        -0.63798948327222038,-0.021960985394712317,0.0,0.0,0.0,0.0,0.0,0.0,1.0,0.0,0.0,-0.0,-0.0,-0.0,-0.0,-0.0,
        -0.0,-1.0,-0.0,0.62490021645747618,0.58505858013174883,0.027072082181883242,0.027610578309122807,
        0.026708907388227909,-0.37854052611351124,-0.027072082181883242,-0.026708907388227909,0.0,0.0,0.0,0.0,0.0,
        0.0,0.0,0.0,-0.0,-0.0,-0.0,-0.0,-0.0,-0.0,-1.0,-0.0,0.027265477962947069,0.55566222109490582,
        0.63798667601923609,0.029437135799321879,0.62488169574462793,-0.55566181651356428,-0.023469887537635192,
        -0.62488169574462793,-0.63798609648432814,0.0,0.0,0.0,0.0,0.0,0.0,1.0,0.0,-0.0,-0.0,-0.0,-0.0,-0.0,-0.0,
        -1.0,-0.0,0.63800507768378822,0.027011667529779945,0.027541181508898387,0.026637267215644224,
        -0.45692709004827581,-0.027011667529779945,-0.58505858013174894,-0.027541181508898383,-0.026637267215644224,
        0.0,0.0,0.0,0.0,0.0,0.0,0.0,0.0,-0.0,-0.0,-0.0,-0.0,-0.0,-0.0,-1.0,-0.0,0.026352061912650541,
        0.55566389422834717,0.62488507878410182,0.637989575133729,-0.55566389422834717,-0.02598312883534095,
        -0.62488507878410182,-0.0294371357993219,-0.63798957513372911,0.0,0.0,0.0,0.0,0.0,0.0,1.0,0.0,-0.0,-0.0,
        -0.0,-0.0,-0.0,-0.0,-1.0,-0.0,-0.55566424910285672,-0.027034185307057621,0.70224208707170055,
        0.024752136540096732,0.70251617195999394,0.022319435462106595,0.0,0.0,0.0,0.0,0.0,0.0,0.0,0.0,-0.0,-0.0,
        -0.0,-0.0,-0.0,-0.0,-1.0,-0.0,-0.70226225634217332,-0.3785405261135113,-0.70163518723474272,
        0.027105602758215112,0.027648865450003536,0.026748274296612785,-0.027105602758215112,-0.027648865450003533,
        -0.026748274296612785,0.0,0.0,0.0,0.0,0.0,0.0,1.0,0.0,0.0,0.0,-0.0,-0.0,-0.0,-0.0,-0.0,-0.0,-0.0,
        -0.55566222109490582,0.023637206391576536,0.015100165961297108,-1.0,-0.378540460951947,-0.02764886545000354,
        0.015207454024849647,0.0,0.0,0.0,0.0,0.0,0.0,1.0,0.0,-0.0,-0.0,-0.0,-0.0,-0.0,-0.0,-0.45692709004827575,
        -0.702534060267215,0.027090859530371859,0.70163518723474272,-0.026730661933064313,0.0,0.0,0.0,0.0,0.0,0.0,
        0.0,0.0,-0.0,-0.0,-0.0,-0.0,-0.0,-0.0,-0.0,-0.55566389422834728,0.029709944333287521,-1.0,
        -0.37854017792555505,-0.026748274296612796,0.0,0.0,0.0,0.0,0.0,0.0,1.0,0.0,0.0,-0.0,-0.0,-0.0,-0.0,-0.0,
        -0.0,-0.55566424910285672,0.027034185307057621,-1.0,-0.37851997948504351,0.70317323754735273,
        -0.02240967789339866,0.0,0.0,0.0,0.0,0.0,0.0,0.0,0.0,-0.0,-0.0,-0.0,-0.0,-0.0,-0.0,-0.0,
        -0.55566222109490582,0.027566488177000255,0.70223873149897853,-0.023637206391576546,-0.015100165961297143,
        0.0,0.0,0.0,0.0,0.0,0.0,-0.0,-0.0,-0.0,-0.0,-0.0,-0.0,-1.0,-0.55566389422834728,0.026662833272981429,
        0.70224253943268344,0.70251656286365771,-0.026190122699982339,-0.029709944333287511,0.0,0.0,0.0,0.0,0.0,0.0,
        0.0,-0.0,-0.0,-0.0,-0.0,-0.0,-0.0,-1.0,-0.0,-0.02706527731251647,-0.6248806237808493,-0.023656120772106486,
        0.378519539943052,0.70317018870025627,0.0,0.0,0.0,0.0,0.0,0.0,0.0,0.0,-0.0,-0.0,-0.0,-0.0,-0.0,-0.0,
        -0.02346980199155271,-0.024399835479656976,0.55566129015943833,0.6248806237808493,0.63798497169620461,
        0.01473301981127613,-0.55566129015943833,-0.6248806237808493,-0.63798497169620461,0.0,0.0,0.0,0.0,0.0,0.0,
        1.0,0.0,-0.0,-0.0,-0.0,-0.0,-0.0,-0.0,-0.027011667529779945,-0.63798948327222027,0.456923837504278,
        0.58504518410006956,0.024723646828030479,0.0,0.0,0.0,0.0,0.0,0.0,1.0,0.0,-0.0,-0.0,-0.0,-0.0,-0.0,-0.0,-0.0,
        -0.02598312883534095,-0.021960985394712324,0.63798532239475636,-0.55566147407010114,-0.62488096344828059,
        -0.63798532239475636,0.0,0.0,0.0,0.0,0.0,0.0,1.0,0.0,0.0,0.0,-0.0,-0.0,-0.0,-0.0,-0.0,-0.0,-1.0,
        -0.027034185307057618,0.55566424910285683,0.024752136540096732,-0.70224208707170055,-0.70251617195999394,
        0.0,0.0,0.0,0.0,0.0,0.0,1.0,0.0,-0.0,-0.0,-0.0,-0.0,-0.0,-0.0,-0.0,-0.0,-0.02706527731251647,
        0.62488504774223075,0.024795740829694754,-0.37851997948504357,-0.7031738370963756,0.0,0.0,0.0,0.0,0.0,0.0,
        0.0,-0.0,-0.0,-0.0,-0.0,-0.0,-0.0,-0.0,-0.027011667529779945,0.63798948327222038,0.024723646828030479,
        0.02229166073122648,-0.456923837504278,-0.58504518410006945,0.0,0.0,0.0,0.0,0.0,0.0,0.0,-0.0,-0.0,-0.0,-0.0,
        -0.0,-0.0,-1.0,-0.0,-0.6248822663250807,-0.0276027315782233,-0.58504257002809312,-0.02974148887250478,
        0.37854036201549385,0.023660396850780661,0.0,0.0,0.0,0.0,0.0,0.0,1.0,0.0,-0.0,-0.0,-0.0,-0.0,-0.0,-0.0,
        -0.62488507878410182,-0.026700746627905073,-0.58504502721143925,0.37854017792555522,0.029748443430697026,
        0.0,0.0,0.0,0.0,0.0,0.0,1.0,0.0,-0.0,-0.0,-0.0,-0.0,-0.0,-0.0,-0.62488504774223086,-0.022364818883998015,
        -0.58504518410006956,0.027072082181883231,0.37854107343057747,-0.024805000972806229,0.0,0.0,0.0,0.0,0.0,0.0,
        1.0,0.0,-0.0,-0.0,-0.0,-0.0,-0.0,-0.0,-0.0,-0.58504257002809312,0.027610578309122814,0.37854046095194716,
        -0.023660296965944735,-0.015161281241640749,0.0,0.0,0.0,0.0,0.0,-0.0,-0.0,-0.0,-0.0,-0.0,
        -0.027541181508898383,-0.637986676019236,-0.029685529684818829,0.023621944154890266,0.58504204394174086,0.0,
        0.0,0.0,0.0,0.0,0.0,1.0,0.0,-0.0,-0.0,-0.0,-0.0,-0.0,-0.0,-0.027566488177000262,-0.70251319697861081,
        -0.029709944333287532,0.55566181651356417,0.023637304191565071,-0.70223802681964376,0.0,0.0,0.0,0.0,0.0,0.0,
        1.0,0.0,-0.0,-0.0,-0.0,-0.0,-0.0,-0.0,-0.0,-0.027602731578223291,-0.02974148887250478,0.62488169574462793,
        0.023656120772106482,-0.37851926782050033,-0.70317150299940423,0.0,0.0,0.0,0.0,0.0,-0.0,-0.0,-0.0,-0.0,-0.0,
        -0.027541181508898383,-0.4569226479042604,-0.58504257002809312,-0.029685529684818829,0.637986096484328,
        0.023621944154890266,0.0,0.0,0.0,0.0,0.0,0.0,0.0,-0.0,-0.0,-0.0,-0.0,-0.0,-0.0,-1.0,-0.637989575133729,
        -0.026637267215644217,0.58504502721143936,0.029685529684818846,0.0,0.0,0.0,0.0,0.0,0.0,1.0,0.0,-0.0,-0.0,
        -0.0,-0.0,-0.0,-0.0,-0.63798948327222038,0.027011667529779945,0.58504518410006945,-0.024723646828030466,
        -0.02229166073122648,0.0,0.0,0.0,0.0,0.0,0.0,1.0,0.0,-0.0,-0.0,-0.0,-0.0,-0.0,-0.0,-0.0,-0.637986676019236,
        0.02754118150889838,0.58504257002809312,-0.023621847095687702,-0.015074517622588319,0.0,0.0,0.0,0.0,0.0,
        -0.0,-0.0,-0.0,-0.0,-0.0,-0.637989575133729,0.026637267215644217,0.45692310525642205,0.58504502721143936,
        -0.026171339658097509,-0.029685529684818822,0.0,0.0,0.0,0.0,0.0,0.0,1.0,-0.0,-0.0,-0.0,-0.0,-0.0,-0.0,-0.0,
        -0.026662833272981426,0.55566389422834728,0.029709944333287525,-0.70224253943268344,-0.70251656286365771,
        0.0,0.0,0.0,0.0,0.0,0.0,1.0,0.0,-0.0,-0.0,-0.0,-0.0,-0.0,-0.0,-0.0,-0.026700746627905069,
        0.62488507878410182,0.02974148887250477,-0.37851908394641454,-0.703174067452467,0.0,0.0,0.0,0.0,0.0,-0.0,
        -0.0,-0.0,-0.0,-0.0,-0.026637267215644227,0.637989575133729,0.029685529684818811,-0.456923105256422,
        -0.58504502721143925,0.0,0.0,0.0,0.0,0.0,0.0,0.0,-0.0,-0.0,-0.0,-0.0,-0.0,-0.0,-1.0,0.55566424910285672,
        0.027034185307057621,-0.70224208707170055,-0.024752136540096722,-0.70251617195999394,-0.022319435462106609,
        0.0,0.0,0.0,0.0,0.0,0.0,1.0,0.0,-0.0,-0.0,-0.0,-0.0,-0.0,-0.0,-0.0,-0.0,0.37851943317454484,
        0.70226225634217332,0.027098793108292794,-0.70318478827029374,-0.02674010789169564,0.0,0.0,0.0,0.0,0.0,0.0,
        0.0,-0.0,-0.0,-0.0,-0.0,-0.0,-0.0,-0.0,-0.0,0.55566222109490582,0.027566488177000255,-0.023637206391576546,
        -0.70223873149897853,-0.70251319697861081,-0.015100165961297143,0.0,0.0,0.0,0.0,0.0,-0.0,-0.0,-0.0,-0.0,
        -0.0,-0.0,0.45692709004827575,0.7025340602672151,0.37854052611351124,0.70318478827029385,
        0.027105602758215112,0.027648865450003536,0.026748274296612785,-0.027105602758215112,-0.026748274296612785,
        0.0,0.0,0.0,0.0,0.0,0.0,0.0,0.0,-0.0,-0.0,-0.0,-0.0,-0.0,-0.0,-1.0,-0.0,-0.0,0.55566389422834728,
        0.026662833272981429,-0.026190122699982339,-0.70224253943268344,-0.029709944333287511,-0.70251656286365771,
        0.0,0.0,0.0,0.0,0.0,0.0,1.0,-0.0,-0.0,-0.0,-0.0,-0.0,-0.0,-0.0,-0.0,0.02706527731251647,0.62488504774223075,
        -0.37851997948504357,-0.024795740829694744,-0.7031738370963756,-0.022364818883998022,0.0,0.0,0.0,0.0,0.0,
        -0.0,-0.0,-0.0,-0.0,-0.0,-0.0,0.02346980199155272,0.024399835479656965,0.55566129015943833,
        0.6248806237808493,0.63798497169620461,-0.55566129015943833,-0.6248806237808493,-0.63798497169620461,
        -0.014733019811276159,0.0,0.0,0.0,0.0,0.0,0.0,-0.0,-0.0,-0.0,-0.0,-0.0,-0.0,-1.0,-0.0,0.027011667529779945,
        0.63798948327222038,-0.456923837504278,-0.58504518410006945,-0.024723646828030469,-0.02229166073122648,0.0,
        0.0,0.0,0.0,0.0,0.0,0.0,-0.0,-0.0,-0.0,-0.0,-0.0,-0.0,-1.0,-0.0,0.02598312883534095,0.021960985394712324,
        0.63798532239475636,-0.55566147407010114,-0.029307880059563592,0.0,0.0,0.0,0.0,0.0,0.0,1.0,-0.0,-0.0,-0.0,
        -0.0,-0.0,-0.0,-0.0,0.6248822663250807,0.027602731578223294,-0.37851936679972537,-0.023656021236335204,
        -0.703171917764931,-0.01515082442675411,0.0,0.0,0.0,0.0,-0.0,-0.0,-0.0,-0.0,0.62488507878410182,
        0.58504502721143936,0.026708907388227905,-0.37854017792555511,-0.026218970645527549,-0.029748443430697016,
        0.0,0.0,0.0,0.0,0.0,0.0,-0.0,-0.0,-0.0,-0.0,-0.0,-0.0,-1.0,-0.0,0.02754118150889838,0.63798667601923609,
        -0.4569226479042604,-0.023621847095687692,-0.585042570028093,-0.015074517622588279,0.0,0.0,0.0,0.0,0.0,0.0,
        -0.0,-0.0,-0.0,-0.0,-0.0,-0.0,-1.0,0.63798957513372911,0.026637267215644217,-0.456923105256422,
        -0.026171339658097509,-0.58504502721143925,-0.029685529684818822,0.0,0.0,0.0,0.0,0.0,0.0,-0.0,-0.0,-0.0,
        -0.0,-0.0,-0.0,-1.0,-0.0,-0.702236447861886,-0.37854073327939103,-0.023682030674840704,
        -0.00016424244292451563,0.015216927320390218,0.0,0.0,0.0,0.0,0.0,0.0,1.0,0.0,0.0,-0.0,-0.0,-0.0,-0.0,-0.0,
        -0.0,-0.55566129015943833,-0.023637206391576532,-0.024752136540096732,0.702236447861886,
        0.015109647396991065,0.0,0.0,0.0,0.0,0.0,0.0,-0.0,-0.0,-0.0,-0.0,-0.0,-1.0,-0.45692383750427795,
        -0.70251617195999394,-0.37854107343057741,-0.027105602758215115,0.024849423695496659,0.0,0.0,0.0,0.0,0.0,
        0.0,1.0,0.0,0.0,-0.0,-0.0,-0.0,-0.0,-0.0,-0.0,-0.0,-0.55566181651356428,0.023637304191565081,-1.0,
        -0.015196990314225767,-0.37854036201549374,-0.00027130052193601533,-3.3862997711630647E-5,0.0,0.0,0.0,0.0,
        0.0,0.0,1.0,0.0,0.0,-0.0,-0.0,-0.0,-0.0,-0.0,-0.0,-0.45692310525642194,-0.70251656286365771,
        -0.37854017792555505,-0.70317346814293025,0.026748274296612796,-0.026245744732980112,-0.029783569798323813,
        0.0,0.0,0.0,0.0,0.0,0.0,1.0,0.0,-0.0,-0.0,-0.0,-0.0,-0.0,-0.0,-0.0,-0.55566129015943833,
        0.023637206391576536,0.024752136540096725,0.702236447861886,-0.015109647396991065,0.0,0.0,0.0,0.0,0.0,0.0,
        -0.0,-0.0,-0.0,-0.0,-0.0,-0.0,-1.0,-0.0,-0.55566181651356428,0.029709944333287493,0.70223802681964376,
        0.7025125679269647,-0.023637304191565092,0.0,0.0,0.0,0.0,0.0,0.0,0.0,-0.0,-0.0,-0.0,-0.0,-0.0,-0.0,-1.0,
        -0.0,-0.027072082181883235,-0.58504518410006945,-0.70317383709637549,0.37854107343057752,
        0.024805000972806222,0.0,0.0,0.0,0.0,0.0,0.0,1.0,0.0,-0.0,-0.0,-0.0,-0.0,-0.0,-0.0,-0.0,
        -0.024723646828030497,-0.63798497169620449,-0.023621944154890263,0.5850406398453023,0.0,0.0,0.0,0.0,0.0,0.0,
        1.0,0.0,0.0,-0.0,-0.0,-0.0,-0.0,-0.0,-0.0,-0.023469887537635181,-3.2815184442066549E-5,0.55566088508118927,
        0.62488005247477207,0.63798439140804353,-0.55566088508118927,-0.62488005247477207,-0.63798439140804353,0.0,
        0.0,0.0,0.0,0.0,0.0,1.0,0.0,0.0,0.0,-0.0,-0.0,-0.0,-0.0,-0.0,-0.0,-1.0,-0.024752136540096736,
        -0.70251116957088389,-0.023637304191565078,0.55566088508118927,-0.7022357422084774,0.0,0.0,0.0,0.0,0.0,0.0,
        1.0,0.0,0.0,-0.0,-0.0,-0.0,-0.0,-0.0,-0.0,-0.0,-0.024795740829694764,-0.023656120772106475,
        0.624880052474772,-0.37851953994305221,-0.70317018870025627,0.0,0.0,0.0,0.0,0.0,0.0,-0.0,-0.0,-0.0,-0.0,
        -0.0,-0.023621847095687688,-0.024723646828030497,0.63798497169620461,0.015083998191321592,
        -0.45692247149286119,-0.58504116656491612,0.0,0.0,0.0,0.0,0.0,0.0,0.0,-0.0,-0.0,-0.0,-0.0,-0.0,-0.0,
        -0.023621944154890259,-3.3598535051162514E-5,0.0050973150136454475,-0.45692225021991206,
        -0.58504063984530219,0.0,0.0,0.0,0.0,0.0,0.0,0.0,0.0,-0.0,-0.0,-0.0,-0.0,-0.0,-0.0,-1.0,
        -0.027098793108292798,0.37851997948504373,0.70224208707170055,-0.70317323754735284,0.0,0.0,0.0,0.0,0.0,0.0,
        0.0,-0.0,-0.0,-0.0,-0.0,-0.0,-0.0,-0.0,-0.0,-0.027090859530371859,-0.023672783354342114,0.4569224714928613,
        0.70251116957088389,0.015195086849570095,-0.70160323232532973,0.0,0.0,0.0,0.0,0.0,0.0,-0.0,-0.0,-0.0,-0.0,
        -0.0,-0.0,-0.0,-0.027072082181883235,0.58504518410006934,0.024805000972806222,0.022374380992921029,
        -0.37854107343057752,0.0,0.0,0.0,0.0,0.0,0.0,0.0,-0.0,-0.0,-0.0,-0.0,-0.0,-0.0,-1.0,-0.0,
        -0.58504502721143925,-0.70317406745246691,0.026708907388227905,0.37854017792555522,-0.026218970645527549,
        -0.029748443430697016,0.0,0.0,0.0,0.0,0.0,0.0,1.0,-0.0,-0.0,-0.0,-0.0,-0.0,-0.0,-0.0,-0.585041166564916,
        0.023660296965944742,0.024805000972806225,0.37854073327939119,-0.015170756558948674,0.0,0.0,0.0,0.0,0.0,
        -0.0,-0.0,-0.0,-0.0,-1.0,-0.0,-0.62488169574462793,-0.58504204394174075,0.029748443430697009,
        0.37854036201549396,-0.023660396850780658,0.0,0.0,0.0,0.0,0.0,0.0,1.0,-0.0,-0.0,-0.0,-0.0,-0.0,-0.0,-0.0,
        -0.027631856629547157,0.4569226479042604,0.70251319697861081,0.023672783354342117,0.015185611969090922,
        -0.70160605506782658,0.0,0.0,0.0,0.0,0.0,-0.0,-0.0,-0.0,-0.0,-0.0,-0.0,-0.0,-0.027610578309122811,
        -0.02974844343069703,0.58504204394174075,0.023660396850780651,-0.37854036201549374,0.0,0.0,0.0,0.0,0.0,0.0,
        0.0,-0.0,-0.0,-0.0,-0.0,-0.0,-0.0,-1.0,-0.63798497169620449,0.0236218470956877,0.024723646828030469,
        0.58504116656491612,-0.015083998191321633,0.0,0.0,0.0,0.0,0.0,-0.0,-0.0,-0.0,-0.0,-1.0,-0.0,
        0.026171339658097509,0.022291660731226463,0.58504146009743707,-0.0050973150136454448,0.023621944154890263,
        0.45692225021991223,0.0,0.0,0.0,0.0,0.0,0.0,1.0,-0.0,-0.0,-0.0,-0.0,-0.0,-0.0,-0.0,-0.0,-0.637986096484328,
        0.029685529684818798,0.45692242688405121,0.58504204394174086,-0.02362194415489029,0.0,0.0,0.0,0.0,0.0,0.0,
        1.0,-0.0,-0.0,-0.0,-0.0,-0.0,-0.0,-0.0,-0.026730661933064309,0.45692310525642194,0.70251656286365771,
        0.029768291394636794,-0.70161080096520145,0.0,0.0,0.0,0.0,0.0,0.0,0.0,-0.0,-0.0,-0.0,-0.0,-0.0,-0.0,-0.0,
        -0.026708907388227905,0.58504502721143925,0.029748443430697019,-0.378540177925555,0.0,0.0,0.0,0.0,0.0,0.0,
        0.0,-0.0,-0.0,-0.0,-0.0,-0.0,-0.0,-1.0,0.4569238375042779,0.027090859530371863,0.70251617195999394,
        0.37854107343057747,-0.024849423695496649,-0.022419246501157553,0.0,0.0,0.0,0.0,0.0,0.0,0.0,-0.0,-0.0,-0.0,
        -0.0,-0.0,-0.0,-1.0,-0.0,-0.0,0.55566147407010114,0.026190122699982339,0.0223194354621066,
        -0.70223692196481524,-0.029647784654081327,-0.70251158235928435,0.0,0.0,0.0,0.0,0.0,1.0,-0.0,-0.0,-0.0,-0.0,
        -0.0,-0.0,-0.0,-0.0,0.70224253943268344,0.378540177925555,0.70161080096520145,0.026748274296612796,
        -0.029783569798323813,0.0,0.0,0.0,0.0,0.0,0.0,-0.0,-0.0,-0.0,-0.0,-0.0,-0.0,-1.0,-0.0,-0.0,
        0.45692264790426035,0.027631856629547154,0.70251319697861092,-0.023672783354342128,-0.70160605506782658,
        -0.015185611969090976,0.0,0.0,0.0,0.0,-0.0,-0.0,-0.0,-0.0,-0.0,-0.0,0.55566181651356428,
        0.029709944333287493,-0.023637304191565092,-0.70223802681964376,-0.7025125679269647,0.0,0.0,0.0,0.0,0.0,0.0,
        1.0,-0.0,-0.0,-0.0,-0.0,-0.0,-0.0,-0.0,-0.0,0.45692310525642188,0.70251656286365771,0.026730661933064316,
        -0.026234238763943405,-0.70161080096520145,-0.029768291394636756,0.0,0.0,0.0,0.0,0.0,-0.0,-0.0,-0.0,-0.0,
        -0.0,-0.0,-0.0,0.027072082181883235,0.58504518410006934,-0.37854107343057752,-0.024805000972806211,
        -0.022374380992921029,0.0,0.0,0.0,0.0,0.0,0.0,0.0,-0.0,-0.0,-0.0,-0.0,-0.0,-0.0,-1.0,-0.0,0.026213688698745,
        0.62488096344828059,0.022364818883998026,-0.3785195589565879,-0.029687807671632122,-0.70317085483536168,0.0,
        0.0,0.0,0.0,-0.0,-0.0,-0.0,-0.0,-0.0,-0.0,0.023469887537635188,0.00012845955535528616,0.55566088508118927,
        0.62488005247477207,0.63798439140804353,-0.55566088508118927,-0.62488005247477207,-0.63798439140804353,0.0,
        0.0,0.0,0.0,0.0,0.0,1.0,0.0,-0.0,-0.0,-0.0,-0.0,-0.0,-0.0,-1.0,-0.0,-0.0,0.585042570028093,
        0.027610578309122811,-0.37854046095194716,-0.023660296965944742,-0.015161281241640751,0.0,0.0,0.0,0.0,0.0,
        0.0,-0.0,-0.0,-0.0,-0.0,-0.0,-0.0,-1.0,0.62488169574462793,0.029741488872504766,-0.3785192678205006,
        -0.023656120772106493,-0.70317150299940423,0.0,0.0,0.0,0.0,0.0,0.0,-0.0,-0.0,-0.0,-0.0,-0.0,-0.0,-0.0,
        0.029685529684818805,0.637986096484328,-0.45692242688405116,-0.02362194415489028,-0.58504204394174075,0.0,
        0.0,0.0,0.0,0.0,0.0,-0.0,-0.0,-0.0,-0.0,-0.0,-0.0,-1.0,-0.0,-0.55566088508118927,-0.023637304191565081,
        -0.015109647396991093,0.7022357422084774,0.0,0.0,0.0,0.0,0.0,0.0,0.0,0.0,0.0,-0.0,-0.0,-0.0,-0.0,-0.0,-0.0,
        -1.0,-0.37854107343057741,-0.0015613656062954475,0.027105602758215108,-0.02484942369549667,
        -0.02241924650115756,0.0,0.0,0.0,0.0,0.0,0.0,1.0,0.0,0.0,-0.0,-0.0,-0.0,-0.0,-0.0,-0.0,-0.0,
        -0.37854046095194693,-0.70317131702755065,0.027648865450003536,-0.023682030674840704,-0.015207454024849647,
        0.0,0.0,0.0,0.0,0.0,0.0,-0.0,-0.0,-0.0,-0.0,-0.0,-0.702236447861886,0.024840157186683216,
        -0.37854073327939092,0.023682030674840707,0.0001642424429245156,-0.015216927320390209,0.0,0.0,0.0,0.0,0.0,
        -0.0,-0.0,-0.0,-0.0,-1.0,-0.0,-0.45692242688405105,-0.7025125679269647,0.02976829139463676,
        -0.37854036201549374,0.00027130052193601533,-0.023682132033406258,0.0,0.0,0.0,0.0,0.0,0.0,1.0,0.0,-0.0,-0.0,
        -0.0,-0.0,-0.0,-0.0,-0.0,-0.55566088508118927,0.023637304191565085,0.029647784654081352,0.7022357422084774,
        0.70251053960656562,0.0,0.0,0.0,0.0,0.0,0.0,0.0,-0.0,-0.0,-0.0,-0.0,-0.0,-0.0,-1.0,-0.0,-0.0,
        -0.37851926782050049,-0.70223802681964376,0.029776610295742294,0.70317090201170729,-0.023677852874347757,
        0.0,0.0,0.0,0.0,0.0,0.0,0.0,-0.0,-0.0,-0.0,-0.0,-0.0,-0.0,-0.58504116656491612,-0.024805000972806236,
        -0.70317060420331423,-0.023660396850780658,-0.0015608627398630522,0.3785406342380947,0.0,0.0,0.0,0.0,0.0,
        0.0,1.0,0.0,0.0,-0.0,-0.0,-0.0,-0.0,-0.0,-0.0,-0.023660296965944735,-0.024805000972806239,
        0.58504116656491578,0.015170756558948695,-0.37854073327939125,0.0,0.0,0.0,0.0,0.0,0.0,0.0,-0.0,-0.0,-0.0,
        -0.0,-0.0,-0.0,-3.3895386058154954E-5,0.0,-1.0,-0.023682030674840707,0.37854073327939108,
        0.0030612231608958297,0.0,0.0,0.0,0.0,0.0,0.0,0.0,-0.0,-0.0,-0.0,-0.0,-0.0,-0.0,-0.0,-0.023660396850780651,
        -3.37922497221569E-5,0.0053104157804372727,-0.37854063423809481,0.0,0.0,0.0,0.0,0.0,0.0,0.0,0.0,-0.0,-0.0,
        -0.0,-0.0,-0.0,-0.0,-1.0,-0.027105602758215112,0.37854107343057758,0.0030612088654606811,
        0.024849423695496673,0.02241924650115756,0.0,0.0,0.0,0.0,0.0,0.0,0.0,-0.0,-0.0,-0.0,-0.0,-0.0,-0.0,-1.0,
        -0.0,-0.0,0.026218970645527546,0.022374380992921033,0.37854065319208563,-0.00531041578043727,
        0.023660396850780661,0.0,0.0,0.0,0.0,0.0,0.0,1.0,-0.0,-0.0,-0.0,-0.0,-0.0,-0.0,-0.0,-0.0,
        -0.015185611969090872,0.45692242688405116,0.7025125679269647,0.023672883991351843,-0.00027130052193601566,
        -3.3862997711630437E-5,0.3785403620154939,0.0,0.0,0.0,0.0,0.0,0.0,0.0,-0.0,-0.0,-0.0,-0.0,-0.0,-0.0,-1.0,
        -0.0,-0.027648865450003536,0.378540460951947,0.70160605506782647,0.0236820306748407,0.015207454024849618,
        0.0,0.0,0.0,0.0,0.0,0.0,-0.0,-0.0,-0.0,-0.0,-0.0,-0.0,-1.0,-0.0,-0.026748274296612789,0.37854017792555505,
        0.70161080096520156,0.029783569798323847,0.0,0.0,0.0,0.0,0.0,0.0,0.0,-0.0,-0.0,-0.0,-0.0,-0.0,-0.0,-1.0,
        -0.0,0.45692249061308471,0.026234238763943405,0.70251158235928435,0.022398709579893369,-0.70160383989347,
        -0.029720779304182428,0.0,0.0,0.0,0.0,-0.0,-0.0,-0.0,-0.0,-0.0,-0.0,-0.0,-0.0,0.55566088508118927,
        0.023637304191565085,0.029647784654081352,-0.7022357422084774,-0.70251053960656573,0.0,0.0,0.0,0.0,0.0,0.0,
        1.0,-0.0,-0.0,-0.0,-0.0,-0.0,-0.0,-0.0,-0.0,-0.0,0.027648865450003536,-1.0,0.37851926782050049,
        0.70223802681964376,0.029776610295742294,-0.023677852874347757,0.0,0.0,0.0,0.0,0.0,0.0,-0.0,-0.0,-0.0,-0.0,
        -0.0,-0.0,-0.0,-0.0,0.45692242688405105,0.02976829139463676,0.7025125679269647,-0.023672883991351864,
        -0.70160519311325342,0.0,0.0,0.0,0.0,0.0,-0.0,-0.0,-0.0,-0.0,-0.0,-0.0,-0.0,0.62488005247477207,
        0.023660396850780661,0.0053104157804372719,3.3792249722156905E-5,-0.3785406342380947,0.0,0.0,0.0,0.0,0.0,
        0.0,-0.0,-0.0,-0.0,-0.0,-0.0,-0.0,-1.0,-0.0,-0.0,0.023621944154890277,0.00012982492179038625,
        0.0050973150136454466,-0.45692225021991212,-0.5850406398453023,0.0,0.0,0.0,0.0,0.0,0.0,-0.0,-0.0,-0.0,-0.0,
        -0.0,-0.0,-1.0,-0.0,-0.0,0.58504204394174064,0.029748443430697026,0.70317150299940412,0.015161281241640776,
        -0.37854036201549396,-0.023660396850780654,0.0,0.0,0.0,0.0,0.0,0.0,-0.0,-0.0,-0.0,-0.0,-0.0,-0.0,-1.0,-0.0,
        -0.378519539943052,-0.023677852874347757,-0.0046218484590718626,-3.3872049431451388E-5,0.70316958685172248,
        0.0,0.0,0.0,0.0,0.0,0.0,0.0,0.0,0.0,-0.0,-0.0,-0.0,-0.0,-0.0,-0.0,-0.37854065319208546,
        9.9046128627942282E-5,-0.029739987791949973,0.0,0.0,0.0,0.0,0.0,1.0,0.0,0.0,0.0,-0.0,-0.0,-0.0,-0.0,-0.0,
        -0.0,-0.0,-0.37851953994305204,0.00013032533543202578,-0.0030612242404972137,0.023682132033406265,
        0.00013036341924922685,0.0,0.0,0.0,0.0,0.0,0.0,1.0,0.0,-0.0,-0.0,-0.0,-0.0,-0.0,-0.0,-0.0,-0.0,
        -0.45692225021991212,-0.0030912635403395824,0.02367288399135186,0.70160236926968877,0.0,0.0,0.0,0.0,0.0,0.0,
        0.0,-0.0,-0.0,-0.0,-0.0,-0.0,-0.0,-0.0,-0.0,0.45692225021991212,0.02367288399135186,0.00013027879750649216,
        0.003091263540339582,-0.70160236926968877,0.0,0.0,0.0,0.0,0.0,-0.0,-0.0,-0.0,-0.0,-0.0,-0.0,-0.0,-0.0,
        0.378519539943052,0.0046218484590718626,0.023682132033406265,3.389538605815513E-5,0.0,0.0,0.0,0.0,0.0,0.0,
        -0.0,-0.0,-0.0,-0.0,-0.0,-0.0,-1.0,-0.0,-0.0,-0.0,-0.37854063423809459,-0.023682132033406265,
        -0.001561372566461268,-3.389538605815513E-5,0.0,0.0,0.0,0.0,0.0,0.0,1.0,0.0,0.0,0.0,-0.0,-0.0,-0.0,-0.0,
        -0.0,-0.0,0.047678521358187322,0.55787204405389446,0.048825402242851326,0.62654723292970194,
        0.047286920841764508,0.63943141348019983,-0.047678521358187322,-0.55787204405389446,-0.048825402242851333,
        -0.62654723292970194,-0.047286920841764508,-0.63943141348019983,0.0,0.0,0.0,0.0,0.0,0.0,0.0,1.0,0.0,0.0,
        -0.0,-0.0,-0.0,-0.0,-0.0,-0.0,-0.0,-1.0,-0.047678521358187315,0.557872509055183,0.044288901125137163,
        0.62654217515979649,0.040021361425923357,0.63942545184526778,-0.557872509055183,-0.62654217515979649,
        -0.63942545184526778,0.0,0.0,0.0,0.0,0.0,0.0,1.0,0.0,0.0,-0.0,-0.0,-0.0,-0.0,-0.0,-0.0,-0.0,-1.0,
        -0.55787204405389446,0.047942655141777091,0.049117799127055072,0.702875228655225,0.0475823178492932,
        0.70295568967385469,-0.047942655141777091,-0.049117799127055078,-0.04758231784929319,0.0,0.0,0.0,0.0,0.0,
        0.0,0.0,0.0,0.0,-0.0,-0.0,-0.0,-0.0,-0.0,-0.0,-0.0,-1.0,-0.048825402242851333,-0.55787171658183987,
        -0.63942424475811355,-0.052452304750527382,0.041298149353625656,0.557871608027596,0.62654080641868248,
        0.63942401877909183,-0.62654080641868248,0.0,0.0,0.0,0.0,0.0,0.0,0.0,1.0,0.0,-0.0,-0.0,-0.0,-0.0,-0.0,-0.0,
        -1.0,-0.626547232929702,-0.047984758880296075,-0.04763006590676714,-0.58732864799299578,
        0.047993536136706469,0.38140732638781982,0.049174830154444668,0.047640075741515714,0.0,0.0,0.0,0.0,0.0,0.0,
        0.0,1.0,0.0,-0.0,-0.0,-0.0,-0.0,-0.0,-0.0,-0.0,-0.047286920841764508,0.045941301434432633,
        0.55787142569916037,0.052452304750527444,0.62654193427993921,0.639425363845251,-0.55787142569916037,
        -0.62654193427993921,-0.639425363845251,0.0,0.0,0.0,0.0,0.0,0.0,0.0,1.0,0.0,-0.0,-0.0,-0.0,-0.0,-0.0,-0.0,
        -1.0,-0.63943141348019983,0.047934264404490834,0.45972838564453733,0.0491093915715111,0.58732864799299578,
        0.04757405784581345,-0.047934264404490834,-0.0491093915715111,-0.04757405784581345,0.0,0.0,0.0,0.0,0.0,0.0,
        0.0,1.0,0.0,-0.0,-0.0,-0.0,-0.0,-0.0,-0.0,-0.0,0.047678521358187315,0.557872509055183,0.62654217515979649,
        0.63942545184526778,-0.557872509055183,-0.044288901125137184,-0.62654217515979649,-0.04002136142592335,
        -0.63942545184526778,0.0,0.0,0.0,0.0,0.0,0.0,0.0,1.0,0.0,-0.0,-0.0,-0.0,-0.0,-0.0,-0.0,-1.0,-0.0,
        0.55787204405389446,0.047942655141777091,0.049117799127055072,0.0475823178492932,-0.047942655141777091,
        -0.049117799127055078,-0.702875228655225,-0.04758231784929319,-0.70295568967385469,0.0,0.0,0.0,0.0,0.0,0.0,
        0.0,1.0,0.0,-0.0,-0.0,-0.0,-0.0,-0.0,-0.0,-0.0,-0.0,0.048825402242851333,0.05245230475052743,
        0.557871608027596,0.62654080641868248,0.63942401877909183,-0.041298149353625628,-0.557871608027596,
        -0.63942401877909183,0.0,0.0,0.0,0.0,0.0,0.0,1.0,0.0,-0.0,-0.0,-0.0,-0.0,-0.0,-0.0,-0.0,-1.0,
        0.626547232929702,0.047984758880296075,0.047630065906767147,0.58732864799299578,0.049174830154444668,
        -0.047993536136706469,-0.38140732638781982,-0.049174830154444675,-0.047640075741515707,0.0,0.0,0.0,0.0,0.0,
        0.0,0.0,0.0,-0.0,-0.0,-0.0,-0.0,-0.0,-0.0,-0.0,-1.0,0.047286920841764508,0.55787142569916037,
        0.62654193427993921,0.639425363845251,-0.045941301434432633,-0.55787142569916037,-0.052452304750527472,
        -0.62654193427993921,-0.639425363845251,0.0,0.0,0.0,0.0,0.0,0.0,1.0,0.0,-0.0,-0.0,-0.0,-0.0,-0.0,-0.0,-0.0,
        -1.0,0.63943141348019983,0.047934264404490834,0.0491093915715111,0.04757405784581345,-0.047934264404490834,
        -0.45972838564453733,-0.0491093915715111,-0.58732864799299578,-0.04757405784581345,0.0,0.0,0.0,0.0,0.0,0.0,
        0.0,0.0,-0.0,-0.0,-0.0,-0.0,-0.0,-0.0,-0.0,-1.0,-0.047942655141777091,-0.557872509055183,
        0.044607913288060984,0.70286297549379462,0.040334527208629158,0.70294446596883164,0.0,0.0,0.0,0.0,0.0,0.0,
        0.0,0.0,-0.0,-0.0,-0.0,-0.0,-0.0,-0.0,-0.0,-1.0,-0.04428890112513717,-0.041298149353625621,
        -0.052879406986409215,0.557871950150472,0.62654033525020214,0.6394234093758725,-0.557871950150472,
        -0.62654033525020214,-0.6394234093758725,0.0,0.0,0.0,0.0,0.0,0.0,0.0,1.0,0.0,0.0,-0.0,-0.0,-0.0,-0.0,-0.0,
        -0.0,-1.0,-0.047984758880296068,0.38139322558672084,0.70313339581753054,-0.0,-0.041515729018567704,
        -0.62654033525020214,0.70313108620605158,0.0,0.0,0.0,0.0,0.0,0.0,0.0,0.0,-0.0,-0.0,-0.0,-0.0,-0.0,-0.0,
        -0.045941301434432633,-0.040021361425923357,0.55787198584888142,0.0528794069864092,-0.63942378652894072,0.0,
        0.0,0.0,0.0,0.0,0.0,0.0,0.0,-0.0,-0.0,-0.0,-0.0,-0.0,-0.0,-1.0,-0.047934264404490841,0.587326232489261,-0.0,
        -0.041479097778282452,-0.6394234093758725,0.0,0.0,0.0,0.0,0.0,0.0,0.0,1.0,0.0,-0.0,-0.0,-0.0,-0.0,-0.0,-0.0,
        -0.047942655141777091,0.557872509055183,-0.0,-0.041486488318378048,0.027677161979573293,
        -0.70294159791647837,0.0,0.0,0.0,0.0,0.0,0.0,1.0,0.0,-0.0,-0.0,-0.0,-0.0,-0.0,-0.0,-0.0,
        -0.047984758880296068,0.62654217515979649,0.044660621016635559,-0.38139322558672084,-0.70313339581753065,
        0.0,0.0,0.0,0.0,0.0,0.0,-0.0,-0.0,-0.0,-0.0,-0.0,-0.0,-0.0,-0.047934264404490841,0.63942545184526778,
        0.0446006835917423,0.040327604063683457,-0.45973364369000819,-0.587326232489261,0.0,0.0,0.0,0.0,0.0,0.0,0.0,
        -0.0,-0.0,-0.0,-0.0,-0.0,-0.0,-0.0,-1.0,-0.55787171658183987,-0.049198241144151271,-0.38141432182325924,
        0.041543427917705961,0.027753531302003462,0.0,0.0,0.0,0.0,0.0,0.0,1.0,0.0,-0.0,-0.0,-0.0,-0.0,-0.0,-0.0,
        -0.381386025829566,-0.702875228655225,0.048014979218259819,0.049198241144151264,0.047663646280299156,
        0.70314122138856006,-0.048014979218259819,-0.049198241144151271,-0.047663646280299156,0.0,0.0,0.0,0.0,0.0,
        0.0,0.0,0.0,-0.0,-0.0,-0.0,-0.0,-0.0,-0.0,-0.55787142569916048,-0.04758231784929319,0.046165728248822986,
        0.052734339992385214,0.70286396678410767,0.0,0.0,0.0,0.0,0.0,0.0,0.0,0.0,-0.0,-0.0,-0.0,-0.0,-0.0,-0.0,-1.0,
        -0.45972838564453744,-0.70295568967385458,0.04765651814247162,-0.048008393947647693,-0.049191105586226781,
        -0.047656518142471613,0.0,0.0,0.0,0.0,0.0,0.0,0.0,1.0,0.0,0.0,-0.0,-0.0,-0.0,-0.0,-0.0,-0.0,-0.0,
        -0.557872509055183,0.0479426551417771,0.70286297549379462,-0.044607913288061025,-0.040334527208629151,0.0,
        0.0,0.0,0.0,0.0,0.0,0.0,0.0,-0.0,-0.0,-0.0,-0.0,-0.0,-0.0,-1.0,-0.0,-0.55787171658183987,
        0.049117799127055085,0.70286143698134129,-0.041486488318378041,-0.027661054311066195,0.0,0.0,0.0,0.0,0.0,
        0.0,0.0,-0.0,-0.0,-0.0,-0.0,-0.0,-0.0,-1.0,-0.55787142569916048,0.04758231784929319,0.70286396678410767,
        0.70294533564091966,-0.046165728248822986,-0.052734339992385255,0.0,0.0,0.0,0.0,0.0,0.0,0.0,-0.0,-0.0,-0.0,
        -0.0,-0.0,-0.0,-0.0,-1.0,-0.049164972356125373,-0.62654101707515264,-0.052779600708881172,
        -0.58732523320298258,0.041521734602731605,0.38141436310945664,0.0,0.0,0.0,0.0,0.0,0.0,0.0,1.0,-0.0,-0.0,
        -0.0,-0.0,-0.0,-0.0,-0.049109391571511091,-0.63942424475811355,-0.052725613098002319,0.041479097778282452,
        0.58732507052489791,0.0,0.0,0.0,0.0,0.0,0.0,0.0,1.0,-0.0,-0.0,-0.0,-0.0,-0.0,-0.0,-0.049117799127055078,
        -0.70294302173702006,-0.052734339992385228,0.557871608027596,0.041486711482857687,-0.70286111061272671,0.0,
        0.0,0.0,0.0,0.0,0.0,0.0,1.0,-0.0,-0.0,-0.0,-0.0,-0.0,-0.0,-0.0,-0.052779600708881172,0.62654080641868259,
        0.041515729018567711,-0.381393060579516,-0.70313207851881332,0.0,0.0,0.0,0.0,0.0,-0.0,-0.0,-0.0,-0.0,-0.0,
        -0.62654193427993921,-0.047630065906767147,-0.58732556690019289,0.38141260703668056,0.052788975072809517,
        0.0,0.0,0.0,0.0,0.0,0.0,0.0,1.0,-0.0,-0.0,-0.0,-0.0,-0.0,-0.0,-0.62654217515979649,-0.040386220026432475,
        -0.587326232489261,0.047993536136706476,0.38141452789755637,-0.044671688889686353,0.0,0.0,0.0,0.0,0.0,0.0,
        0.0,1.0,-0.0,-0.0,-0.0,-0.0,-0.0,-0.0,-0.0,-0.62654101707515253,-0.58732523320298247,0.049174830154444668,
        0.38141432182325907,-0.041521509739207062,-0.027720209169872088,0.0,0.0,0.0,0.0,0.0,-0.0,-0.0,-0.0,-0.0,
        -0.0,-0.62654193427993921,-0.04620090230449761,-0.0527796007088812,-0.58732556690019289,0.0476400757415157,
        0.38141260703668056,0.0,0.0,0.0,0.0,0.0,0.0,1.0,-0.0,-0.0,-0.0,-0.0,-0.0,-0.0,-0.0,-0.047574057845813457,
        -0.639425363845251,0.052725613098002347,0.58732556690019289,0.0,0.0,0.0,0.0,0.0,0.0,0.0,1.0,-0.0,-0.0,-0.0,
        -0.0,-0.0,-0.0,-0.04758231784929319,0.55787142569916037,0.052734339992385269,-0.70286396678410767,
        -0.70294533564091966,0.0,0.0,0.0,0.0,0.0,0.0,0.0,1.0,-0.0,-0.0,-0.0,-0.0,-0.0,-0.0,-0.0,
        -0.04763006590676714,0.62654193427993921,0.052779600708881193,-0.38139130491870232,-0.703133933677141,0.0,
        0.0,0.0,0.0,0.0,-0.0,-0.0,-0.0,-0.0,-0.0,-0.047574057845813457,0.639425363845251,0.04615757913241255,
        0.052725613098002347,-0.45973190050489804,-0.58732556690019289,0.0,0.0,0.0,0.0,0.0,0.0,0.0,-0.0,-0.0,-0.0,
        -0.0,-0.0,-0.0,-1.0,-0.63942545184526778,0.047934264404490834,0.587326232489261,-0.044600683591742338,
        -0.04032760406368343,0.0,0.0,0.0,0.0,0.0,0.0,0.0,1.0,-0.0,-0.0,-0.0,-0.0,-0.0,-0.0,-0.0,
        -0.63942424475811355,0.0491093915715111,0.58732523320298258,-0.041478874690674995,-0.027655051949837254,0.0,
        0.0,0.0,0.0,0.0,-0.0,-0.0,-0.0,-0.0,-0.0,-0.639425363845251,0.047574057845813443,0.58732556690019289,
        -0.04615757913241255,-0.052725613098002382,0.0,0.0,0.0,0.0,0.0,0.0,1.0,-0.0,-0.0,-0.0,-0.0,-0.0,-0.0,-0.0,
        0.047942655141777091,0.557872509055183,-0.044607913288061012,-0.70286297549379462,-0.040334527208629144,
        -0.70294446596883164,0.0,0.0,0.0,0.0,0.0,0.0,0.0,1.0,-0.0,-0.0,-0.0,-0.0,-0.0,-0.0,-0.0,-0.0,
        0.041297934356687133,0.0442889011251372,0.55787205898156167,-0.027381569976781938,-0.63942363589545237,0.0,
        0.0,0.0,0.0,0.0,0.0,0.0,-0.0,-0.0,-0.0,-0.0,-0.0,-0.0,-1.0,-0.0,0.047984758880296068,0.62654217515979649,
        -0.38139322558672084,-0.044660621016635579,-0.040386220026432489,-0.70313339581753065,0.0,0.0,0.0,0.0,0.0,
        -0.0,-0.0,-0.0,-0.0,-0.0,-0.0,0.045941301434432633,0.04002136142592335,0.041298149353625628,
        0.027381569976781941,0.557871950150472,0.62654033525020214,0.6394234093758725,-0.557871950150472,
        -0.6394234093758725,0.0,0.0,0.0,0.0,0.0,0.0,1.0,0.0,-0.0,-0.0,-0.0,-0.0,-0.0,-0.0,-0.0,-1.0,-0.0,
        0.047934264404490841,0.63942545184526778,-0.45973364369000819,-0.044600683591742324,-0.587326232489261,
        -0.040327604063683443,0.0,0.0,0.0,0.0,0.0,0.0,0.0,-0.0,-0.0,-0.0,-0.0,-0.0,-0.0,-1.0,-0.0,
        0.55787171658183987,0.049117799127055085,-0.041486488318378041,-0.70286143698134129,-0.027661054311066195,
        -0.70294302173702006,0.0,0.0,0.0,0.0,0.0,-0.0,-0.0,-0.0,-0.0,-0.0,-0.0,0.381386025829566,
        0.70287522865522511,0.048014979218259819,0.049198241144151264,0.047663646280299156,-0.048014979218259819,
        -0.049198241144151271,-0.047663646280299156,-0.70314122138856006,0.0,0.0,0.0,0.0,0.0,0.0,-0.0,-0.0,-0.0,
        -0.0,-0.0,-0.0,-0.0,-0.0,0.55787142569916048,0.04758231784929319,-0.046165728248822986,
        -0.052734339992385255,-0.70286396678410767,-0.70294533564091966,0.0,0.0,0.0,0.0,0.0,0.0,1.0,-0.0,-0.0,-0.0,
        -0.0,-0.0,-0.0,-0.0,-0.0,0.45972838564453744,0.70295568967385458,0.04765651814247162,-0.048008393947647693,
        -0.70268597089371387,0.0,0.0,0.0,0.0,0.0,0.0,0.0,-0.0,-0.0,-0.0,-0.0,-0.0,-0.0,-0.0,0.049164972356125373,
        0.62654101707515264,-0.041515504461835731,-0.38139301933175634,-0.027709698583410016,-0.70313230364575241,
        0.0,0.0,0.0,0.0,-0.0,-0.0,-0.0,-0.0,0.049109391571511105,0.052725613098002361,0.63942401877909172,
        -0.041479097778282459,-0.45973321032477427,-0.58732507052489791,0.0,0.0,0.0,0.0,0.0,0.0,-0.0,-0.0,-0.0,-0.0,
        -0.0,-0.0,-0.0,-1.0,0.62654193427993921,0.047630065906767147,-0.04620090230449761,-0.38139130491870232,
        -0.052779600708881227,-0.703133933677141,0.0,0.0,0.0,0.0,0.0,0.0,-0.0,-0.0,-0.0,-0.0,-0.0,-0.0,-0.0,
        0.047574057845813457,0.639425363845251,-0.046157579132412557,-0.45973190050489804,-0.052725613098002388,
        -0.58732556690019289,0.0,0.0,0.0,0.0,0.0,0.0,-0.0,-0.0,-0.0,-0.0,-0.0,-0.0,-0.0,-1.0,-0.044696511233766632,
        -0.041537644408465073,-0.38139435220779871,-0.0046455551781967915,0.70313098732427648,0.0,0.0,0.0,0.0,0.0,
        0.0,0.0,0.0,0.0,-0.0,-0.0,-0.0,-0.0,-0.0,-0.0,-0.048014979218259812,-0.38139322558672073,
        -0.70286297549379451,0.04469651123376666,0.70313329820348291,0.0,0.0,0.0,0.0,0.0,0.0,-0.0,-0.0,-0.0,-0.0,
        -0.0,-0.0,-0.046165728248822986,-0.040334527208629165,-0.041486711482857673,-0.55787195015047186,
        0.70285954634074388,0.0,0.0,0.0,0.0,0.0,0.0,0.0,0.0,0.0,-0.0,-0.0,-0.0,-0.0,-0.0,-0.0,-1.0,
        -0.047993536136706476,0.38141452789755642,-0.0,-0.70313131216765046,-0.0415217346027316,
        -0.0053499825507371153,-0.0015656878741349531,0.0,0.0,0.0,0.0,0.0,0.0,0.0,1.0,0.0,-0.0,-0.0,-0.0,-0.0,-0.0,
        -0.0,-0.04615757913241255,-0.040327604063683457,-0.041479097778282452,-0.027671157031094271,
        0.6394234093758725,-0.45973424542066693,-0.58732499879699229,0.0,0.0,0.0,0.0,0.0,0.0,0.0,0.0,-0.0,-0.0,-0.0,
        -0.0,-0.0,-0.0,-1.0,-0.048014979218259812,0.38139322558672073,0.70286297549379451,0.04469651123376666,
        -0.70313329820348291,0.0,0.0,0.0,0.0,0.0,0.0,-0.0,-0.0,-0.0,-0.0,-0.0,-0.0,-0.0,-0.0,-0.047993536136706476,
        0.587326232489261,0.044671688889686333,0.040397149349959804,-0.38141452789755642,0.0,0.0,0.0,0.0,0.0,0.0,
        0.0,-0.0,-0.0,-0.0,-0.0,-0.0,-0.0,-0.0,-1.0,-0.557871608027596,-0.052734339992385235,-0.027661054311066337,
        0.041486711482857694,0.70286111061272671,0.0,0.0,0.0,0.0,0.0,0.0,0.0,0.0,-0.0,-0.0,-0.0,-0.0,-0.0,-0.0,-1.0,
        -0.70286396678410779,-0.047663646280299149,-0.38141260703668067,0.052821149416567043,0.0,0.0,0.0,0.0,0.0,
        0.0,0.0,1.0,0.0,-0.0,-0.0,-0.0,-0.0,-0.0,-0.0,-0.38140732638781988,-0.0015661221639725058,
        0.048023761687426413,0.049208104725552843,0.047673661972528605,-0.048023761687426413,-0.049208104725552849,
        -0.0476736619725286,0.0,0.0,0.0,0.0,0.0,0.0,0.0,1.0,0.0,0.0,-0.0,-0.0,-0.0,-0.0,-0.0,-0.0,-0.0,
        -0.70286297549379451,-0.04042146861842183,-0.38141452789755653,0.048023761687426413,-0.044707585477670696,
        0.0,0.0,0.0,0.0,0.0,0.0,0.0,1.0,0.0,-0.0,-0.0,-0.0,-0.0,-0.0,-0.0,-0.0,-0.70286143698134129,
        -0.38141432182325918,0.049208104725552843,-0.041543427917705954,-0.027753531302003361,0.0,0.0,0.0,0.0,0.0,
        0.0,-0.0,-0.0,-0.0,-0.0,-0.0,-0.38139130491870249,-0.70286396678410779,0.047663646280299149,
        0.70313383642924188,-0.046226776721425993,-0.052811769511494744,0.0,0.0,0.0,0.0,0.0,0.0,0.0,-0.0,-0.0,-0.0,
        -0.0,-0.0,-0.0,-0.38141260703668073,-0.0015661807001885121,0.0003808990881292652,-0.046234063364270737,
        -0.052821149416567105,0.0,0.0,0.0,0.0,0.0,0.0,1.0,0.0,-0.0,-0.0,-0.0,-0.0,-0.0,-0.0,-0.0,
        -0.55787205898156167,0.041486488318378034,0.044607913288061032,-0.02767716197957313,0.0,0.0,0.0,0.0,0.0,0.0,
        0.0,-0.0,-0.0,-0.0,-0.0,-0.0,-0.0,-1.0,-0.0,-0.55787198584888142,-0.38139402411953655,0.046226776721426013,
        0.04042146861842183,0.70313145912642394,-0.053301939043787668,0.0,0.0,0.0,0.0,0.0,0.0,-0.0,-0.0,-0.0,-0.0,
        -0.0,-0.0,-0.0,-0.557871608027596,0.052734339992385269,0.70286111061272671,0.70294271779415229,
        -0.041486711482857687,0.0,0.0,0.0,0.0,0.0,0.0,0.0,-0.0,-0.0,-0.0,-0.0,-0.0,-0.0,-0.0,-1.0,
        -0.052725613098002319,-0.027655051949837452,0.63942401877909172,0.041479097778282452,-0.45973321032477427,
        -0.58732507052489791,0.0,0.0,0.0,0.0,0.0,0.0,0.0,-0.0,-0.0,-0.0,-0.0,-0.0,-0.0,-1.0,-0.052811769511494709,
        0.381393060579516,0.70286111061272671,0.041537644408465066,-0.70313198021515855,0.0,0.0,0.0,0.0,0.0,-0.0,
        -0.0,-0.0,-0.0,-0.0,-0.0,-0.049174830154444661,-0.052788975072809545,0.58732507052489813,
        0.041521734602731612,-0.38141436310945631,0.0,0.0,0.0,0.0,0.0,0.0,0.0,-0.0,-0.0,-0.0,-0.0,-0.0,-0.0,-1.0,
        -0.6265406645097189,0.046200902304497617,0.040386220026432475,0.38139402411953627,0.70313155774868141,
        -0.053264773578912634,0.0,0.0,0.0,0.0,0.0,-0.0,-0.0,-0.0,-0.0,-0.0,-0.0,-0.0,-0.62654080641868248,
        -0.58732507052489791,0.052788975072809559,0.38141436310945637,-0.0415217346027316,0.0,0.0,0.0,0.0,0.0,0.0,
        1.0,-0.0,-0.0,-0.0,-0.0,-0.0,-0.0,-0.0,-0.047663646280299156,0.38139130491870238,0.70286396678410779,
        0.052811769511494681,-0.70313383642924188,0.0,0.0,0.0,0.0,0.0,-0.0,-0.0,-0.0,-0.0,-0.0,-0.0,
        0.45973190050489809,0.70294533564091954,0.052804674695198853,-0.00038089908812926509,0.38141260703668056,
        0.046234063364270724,0.0,0.0,0.0,0.0,0.0,0.0,0.0,-0.0,-0.0,-0.0,-0.0,-0.0,-0.0,-1.0,-0.0,
        -0.047640075741515714,0.58732556690019289,0.046208184541143907,0.0527889750728095,-0.38141260703668045,0.0,
        0.0,0.0,0.0,0.0,0.0,0.0,-0.0,-0.0,-0.0,-0.0,-0.0,-0.0,-1.0,-0.63942378652894072,0.046157579132412543,
        0.040327604063683443,0.587325187651558,-0.053202204406742878,0.0,0.0,0.0,0.0,0.0,0.0,1.0,-0.0,-0.0,-0.0,
        -0.0,-0.0,-0.0,-0.0,-0.63942401877909172,0.052725613098002388,0.5873250705248978,-0.041479097778282417,0.0,
        0.0,0.0,0.0,0.0,0.0,1.0,-0.0,-0.0,-0.0,-0.0,-0.0,-0.0,-0.0,0.046165728248822993,0.55787198584888142,
        0.040334527208629144,0.041486711482857666,-0.70285954634074388,-0.70294129315678422,0.0,0.0,0.0,0.0,0.0,0.0,
        1.0,-0.0,-0.0,-0.0,-0.0,-0.0,-0.0,-0.0,-0.0,-0.0,0.048008393947647693,0.45973364369000813,
        0.70294446596883153,-0.04468906953870326,-0.7026717750678485,-0.040414301735567953,0.0,0.0,0.0,0.0,0.0,0.0,
        -0.0,-0.0,-0.0,-0.0,-0.0,-0.0,-0.0,-0.0,0.044600683591742331,0.041479097778282431,0.053202204406742781,
        0.6394234093758725,-0.58732499879699229,0.0,0.0,0.0,0.0,0.0,0.0,-0.0,-0.0,-0.0,-0.0,-0.0,-0.0,-0.0,-1.0,
        -0.0,0.04620090230449761,0.62654066450971879,0.040386220026432489,-0.38139402411953638,
        -0.053264773578912634,-0.70313155774868152,0.0,0.0,0.0,0.0,-0.0,-0.0,-0.0,-0.0,-0.0,-0.0,
        0.047993536136706476,0.587326232489261,-0.38141452789755642,-0.044671688889686353,-0.040397149349959791,0.0,
        0.0,0.0,0.0,0.0,0.0,0.0,-0.0,-0.0,-0.0,-0.0,-0.0,-0.0,-1.0,-0.0,0.046157579132412557,0.040327604063683437,
        0.63942378652894072,-0.4597340245185435,-0.0532022044067428,-0.58732518765155828,0.0,0.0,0.0,0.0,0.0,-0.0,
        -0.0,-0.0,-0.0,-0.0,-0.0,-0.0,0.557871608027596,0.052734339992385269,-0.041486711482857687,
        -0.70286111061272671,-0.70294271779415229,0.0,0.0,0.0,0.0,0.0,0.0,1.0,-0.0,-0.0,-0.0,-0.0,-0.0,-0.0,-0.0,
        -0.0,0.45973321958975349,0.049191105586226788,0.70294302173702006,-0.041532433509010709,
        -0.70267008402296527,-0.027736669979992645,0.0,0.0,0.0,0.0,-0.0,-0.0,-0.0,-0.0,-0.0,-0.0,
        0.38140732638781988,0.0030799473449444718,0.048023761687426413,0.049208104725552843,0.047673661972528605,
        -0.048023761687426413,-0.049208104725552849,-0.0476736619725286,0.0,0.0,0.0,0.0,0.0,0.0,0.0,0.0,-0.0,-0.0,
        -0.0,-0.0,-0.0,-0.0,-0.0,-1.0,-0.0,0.052779600708881207,0.62654080641868259,-0.0415157290185677,
        -0.38139306057951583,-0.70313207851881332,0.0,0.0,0.0,0.0,0.0,0.0,-0.0,-0.0,-0.0,-0.0,-0.0,-0.0,-0.0,
        0.049174830154444675,0.58732523320298258,-0.041521509739207041,-0.381414321823259,-0.027720209169872008,0.0,
        0.0,0.0,0.0,0.0,0.0,-0.0,-0.0,-0.0,-0.0,-0.0,-0.0,-1.0,0.58732556690019289,0.047640075741515707,
        -0.046208184541143907,-0.38141260703668056,-0.052788975072809566,0.0,0.0,0.0,0.0,0.0,0.0,-0.0,-0.0,-0.0,
        -0.0,-0.0,-0.0,-0.0,-1.0,-0.048023761687426413,-0.38141452789755642,-0.70313329820348291,
        0.044707585477670654,0.0,0.0,0.0,0.0,0.0,0.0,1.0,0.0,0.0,-0.0,-0.0,-0.0,-0.0,-0.0,-0.0,-0.0,
        -0.0414867114828577,-6.14559350203706E-5,0.55787195015047186,-0.70285954634074388,-0.70294129315678422,0.0,
        0.0,0.0,0.0,0.0,0.0,0.0,1.0,0.0,-0.0,-0.0,-0.0,-0.0,-0.0,-0.0,-0.0,-0.041515729018567704,
        -0.027725808084743217,0.62654033525020214,-0.38139435220779894,-0.70313108620605158,0.0,0.0,0.0,0.0,0.0,0.0,
        -0.0,-0.0,-0.0,-0.0,-0.0,-0.044696511233766639,0.70285987351907608,-0.04153764440846508,0.3813943522077986,
        0.0046455551781967924,-0.70313098732427659,0.0,0.0,0.0,0.0,0.0,-0.0,-0.0,-0.0,-0.0,-0.0,-0.0,
        -0.046208184541143921,-0.040397149349959804,0.58732518765155828,-0.041521734602731619,0.0053499825507371188,
        -0.38141565496819624,0.0,0.0,0.0,0.0,0.0,0.0,0.0,0.0,-0.0,-0.0,-0.0,-0.0,-0.0,-0.0,-1.0,
        -0.048023761687426413,0.38141452789755642,0.7026717750678485,0.044707585477670654,0.040432404230908,0.0,0.0,
        0.0,0.0,0.0,0.0,0.0,-0.0,-0.0,-0.0,-0.0,-0.0,-0.0,-0.0,-1.0,-0.0,-0.041521509739207062,
        -0.044671688889686333,0.58732516183395489,0.027736318903840668,-0.3814156136550157,0.0,0.0,0.0,0.0,0.0,0.0,
        0.0,-0.0,-0.0,-0.0,-0.0,-0.0,-0.0,-0.052811769511494695,-0.70286111061272671,-0.027743014678389594,
        -0.38141436310945653,-6.1605929268691053E-5,0.04154365368638769,0.0,0.0,0.0,0.0,0.0,0.0,0.0,1.0,0.0,-0.0,
        -0.0,-0.0,-0.0,-0.0,-0.0,-0.38139306057951616,-0.70286111061272671,0.052811769511494744,0.70313198021515855,
        -0.04153764440846508,0.0,0.0,0.0,0.0,0.0,0.0,0.0,-0.0,-0.0,-0.0,-0.0,-0.0,-0.0,-0.0015662095088587794,1.0,
        -0.0,-0.38139435220779888,0.041537644408465059,0.00023256610403676135,0.0,0.0,0.0,0.0,0.0,0.0,0.0,-0.0,-0.0,
        -0.0,-0.0,-0.0,-0.0,-0.0,-0.38141436310945653,-0.0015661981899676553,0.0004794577441265344,
        -0.041543653686387648,0.0,0.0,0.0,0.0,0.0,0.0,1.0,0.0,-0.0,-0.0,-0.0,-0.0,-0.0,-0.0,-0.0,
        -0.55787195015047186,0.041486711482857659,0.00023216176133703439,0.70285954634074388,0.70294129315678422,
        0.0,0.0,0.0,0.0,0.0,0.0,0.0,-0.0,-0.0,-0.0,-0.0,-0.0,-0.0,-0.0,-1.0,-0.0,0.45973321032477421,
        0.70294271779415229,0.041532658817056131,-0.0004794577441265338,0.38141436310945637,0.0,0.0,0.0,0.0,0.0,0.0,
        0.0,-0.0,-0.0,-0.0,-0.0,-0.0,-0.0,-1.0,-0.0,-0.70313155774868141,0.046208184541143935,0.040397149349959777,
        0.38141532678103607,-0.0053499825507371248,-0.0015656878741349477,0.041521734602731612,0.0,0.0,0.0,0.0,0.0,
        0.0,1.0,-0.0,-0.0,-0.0,-0.0,-0.0,-0.0,-0.0,-0.0,-0.62654033525020214,0.041515729018567704,
        0.053264773578912579,0.38139435220779877,0.70313108620605158,0.0,0.0,0.0,0.0,0.0,0.0,-0.0,-0.0,-0.0,-0.0,
        -0.0,-0.0,-0.0,-0.0,-0.63942340937587239,0.041479097778282424,0.053202204406742795,0.58732499879699218,0.0,
        0.0,0.0,0.0,0.0,0.0,1.0,-0.0,-0.0,-0.0,-0.0,-0.0,-0.0,-0.0,-0.0,0.046220967236855211,0.45973402451854339,
        0.04041430173556794,0.7029419471796341,-0.05329394831239747,-0.70266869475347082,0.0,0.0,0.0,0.0,-0.0,-0.0,
        -0.0,-0.0,-0.0,-0.0,-0.0,-0.0,0.048023761687426413,0.38141452789755642,0.7026717750678485,
        -0.044707585477670675,-0.040432404230907985,0.0,0.0,0.0,0.0,0.0,0.0,0.0,-0.0,-0.0,-0.0,-0.0,-0.0,-0.0,-1.0,
        -0.0,-0.0,0.62654033525020214,-0.0,0.041521509739207055,0.04467168888968636,0.58732516183395489,
        -0.3814156136550157,0.0,0.0,0.0,0.0,0.0,0.0,-0.0,-0.0,-0.0,-0.0,-0.0,-0.0,-1.0,-0.0,0.046208184541143914,
        0.58732518765155806,0.040397149349959791,-0.38141532678103618,-0.053276115903559441,0.0,0.0,0.0,0.0,0.0,
        -0.0,-0.0,-0.0,-0.0,-0.0,-0.0,-0.0,0.049208104725552843,0.38141436310945653,0.00047945774412653418,
        0.0015661981899676573,-0.041543653686387676,0.0,0.0,0.0,0.0,0.0,0.0,-0.0,-0.0,-0.0,-0.0,-0.0,-0.0,-0.0,-1.0,
        -0.0,0.38141260703668067,0.0030800493725469838,0.00038089908812926525,-0.046234063364270724,
        -0.052821149416567063,0.0,0.0,0.0,0.0,0.0,0.0,-0.0,-0.0,-0.0,-0.0,-0.0,-0.0,-0.0,-1.0,-0.0,
        0.052788975072809573,0.5873250705248978,0.027720209169872036,0.70313207851881321,-0.041521734602731585,
        -0.38141436310945664,0.0,0.0,0.0,0.0,0.0,0.0,-0.0,-0.0,-0.0,-0.0,-0.0,-0.0,-0.0,-1.0,-0.041543427917705968,
        -0.38141561365501536,-0.00029424831666778297,-0.0015662085872463908,0.027769643467705708,0.0,0.0,0.0,0.0,
        0.0,0.0,1.0,0.0,0.0,-0.0,-0.0,-0.0,-0.0,-0.0,-0.0,-0.041532658817056138,0.0031055287133001592,
        -0.70266788285587956,0.0,0.0,0.0,0.0,0.0,0.0,1.0,0.0,0.0,-0.0,-0.0,-0.0,-0.0,-0.0,-0.0,-0.0,
        -0.041543427917705961,0.0030801002245625041,-0.00023261598934981646,0.381415654968196,0.0030801017285724173,
        0.0,0.0,0.0,0.0,0.0,0.0,0.0,0.0,-0.0,-0.0,-0.0,-0.0,-0.0,-0.0,-1.0,-0.0,-0.046234063364270724,
        -0.00017791507742684638,0.38141532678103585,0.053313287899267439,0.0,0.0,0.0,0.0,0.0,0.0,0.0,-0.0,-0.0,-0.0,
        -0.0,-0.0,-0.0,-1.0,-0.0,0.04623406336427073,0.38141532678103612,0.003080095298344224,
        0.00017791507742684627,-0.053313287899267488,0.0,0.0,0.0,0.0,0.0,-0.0,-0.0,-0.0,-0.0,-0.0,-0.0,-0.0,-0.0,
        0.041543427917705961,0.00029424831666778313,0.38141565496819613,0.0015662095088587807,0.0,0.0,0.0,0.0,0.0,
        0.0,-0.0,-0.0,-0.0,-0.0,-0.0,-0.0,-0.0,-1.0,-0.0,-0.0,-0.041543653686387669,-0.38141565496819613,
        -6.1661881147355389E-5,-0.0015662095088587807,0.0,0.0,0.0,0.0,0.0,0.0,0.0,1.0,0.0,0.0,-0.0,-0.0,-0.0,-0.0,
        -0.0,-0.0,0.60965291149047529,-0.00028893057593309761,0.45432670979185558,-0.00033174749061995039,
        0.41630255411925293,-0.00034245830389696241,-0.60965291149047529,0.00028893057593309761,
        -0.45432670979185558,0.00033174749061995045,-0.41630255411925293,0.00034245830389696241,0.0,0.0,0.0,0.0,0.0,
        0.0,0.0,0.0,1.0,0.0,-0.0,-0.0,-0.0,-0.0,-0.0,-0.0,-0.0,-0.0,-0.60965291149047518,0.0,
        -1.6889645757588247E-16,9.8644403672779264E-20,-1.2631111769540146E-16,4.5223656320158784E-20,0.0,
        -4.9322201836389632E-20,-4.5223656320158784E-20,0.0,0.0,0.0,0.0,0.0,0.0,0.0,1.0,0.0,-0.0,-0.0,-0.0,-0.0,
        -0.0,-0.0,-0.0,-0.0,0.00028893057593309761,0.60962843737462846,0.45430524726196975,-0.00038816816420182134,
        0.41628290531231787,-0.00039473384869379718,-0.60962843737462846,-0.45430524726196975,-0.41628290531231782,
        0.0,0.0,0.0,0.0,0.0,0.0,0.0,1.0,0.0,-0.0,-0.0,-0.0,-0.0,-0.0,-0.0,-0.0,-0.0,-0.45432670979185558,
        7.4814395651655677E-5,8.7898076503418541E-5,-0.55043530483183312,0.84085614120956309,-7.48192953866797E-5,
        -8.5505485825256925E-5,-8.790393854946284E-5,8.5505485825256979E-5,0.0,0.0,0.0,0.0,0.0,0.0,0.0,0.0,0.0,-0.0,
        -0.0,-0.0,-0.0,-0.0,-0.0,-0.0,0.00033174749061995039,-0.609625471048958,-0.416280549869921,
        0.00030075035944006475,0.60962481916553923,-0.00018417146899711554,0.45430208183095055,0.41628002822785948,
        0.0,0.0,0.0,0.0,0.0,0.0,0.0,0.0,1.0,-0.0,-0.0,-0.0,-0.0,-0.0,-0.0,-0.0,-0.41630255411925293,
        0.75758587834764834,-0.0001318993713365724,0.55043530483183345,-0.00015110237018723787,
        -0.00015561198793193225,0.0001318993713365724,0.00015110237018723792,0.00015561198793193225,0.0,0.0,0.0,0.0,
        0.0,0.0,0.0,0.0,0.0,-0.0,-0.0,-0.0,-0.0,-0.0,-0.0,-0.0,0.00034245830389696241,0.60963041253671413,
        -0.00022788856259313032,0.45430697881955218,-0.00030075035944006486,0.41628450770674136,
        -0.60963041253671413,-0.45430697881955218,-0.41628450770674136,0.0,0.0,0.0,0.0,0.0,0.0,0.0,0.0,1.0,-0.0,
        -0.0,-0.0,-0.0,-0.0,-0.0,-0.0,0.60965291149047518,0.0,9.8644403672779264E-20,4.5223656320158784E-20,0.0,
        1.6889645757588247E-16,-4.9322201836389632E-20,1.2631111769540143E-16,-4.5223656320158784E-20,0.0,0.0,0.0,
        0.0,0.0,0.0,0.0,0.0,0.0,-0.0,-0.0,-0.0,-0.0,-0.0,-0.0,-0.0,-1.0,-0.00028893057593309761,0.60962843737462846,
        0.45430524726196975,0.41628290531231787,-0.60962843737462846,-0.45430524726196975,0.00038816816420182151,
        -0.41628290531231782,0.00039473384869379718,0.0,0.0,0.0,0.0,0.0,0.0,0.0,0.0,1.0,-0.0,-0.0,-0.0,-0.0,-0.0,
        -0.0,-0.0,-0.0,0.45432670979185558,0.55043530483183334,-7.48192953866797E-5,-8.5505485825256925E-5,
        -8.790393854946284E-5,-0.84085614120956309,7.48192953866797E-5,8.790393854946284E-5,0.0,0.0,0.0,0.0,0.0,0.0,
        0.0,0.0,-0.0,-0.0,-0.0,-0.0,-0.0,-0.0,-0.0,-0.0,-0.00033174749061995045,0.609625471048958,
        0.41628054986992108,-0.00030075035944006497,0.45430208183095055,-0.60962481916553923,0.00018417146899711535,
        -0.45430208183095055,-0.41628002822785942,0.0,0.0,0.0,0.0,0.0,0.0,0.0,1.0,-0.0,-0.0,-0.0,-0.0,-0.0,-0.0,
        -0.0,-0.0,0.41630255411925293,-0.0001318993713365724,-0.00015110237018723787,-0.00015561198793193225,
        -0.75758587834764834,0.0001318993713365724,-0.55043530483183345,0.00015110237018723792,
        0.00015561198793193225,0.0,0.0,0.0,0.0,0.0,0.0,0.0,0.0,-0.0,-0.0,-0.0,-0.0,-0.0,-0.0,-0.0,-0.0,
        -0.00034245830389696241,0.60963041253671413,0.45430697881955218,0.41628450770674136,-0.60963041253671413,
        0.00022788856259313032,-0.45430697881955218,0.000300750359440065,-0.41628450770674136,0.0,0.0,0.0,0.0,0.0,
        0.0,0.0,1.0,-0.0,-0.0,-0.0,-0.0,-0.0,-0.0,-0.0,-0.0,-0.60962843737462846,6.6103931646927414E-20,
        1.6888786255250324E-16,3.2847016711299215E-19,1.2630515651810637E-16,1.2285470046927208E-19,0.0,0.0,0.0,0.0,
        0.0,0.0,1.0,0.0,-0.0,-0.0,-0.0,-0.0,-0.0,-0.0,-0.0,-0.0,-1.6889645757588244E-16,-0.840856141209563,
        -5.0906254663616592E-16,-6.6103349467276677E-20,4.9321661480447027E-20,0.0,6.6103349467276677E-20,0.0,0.0,
        0.0,0.0,0.0,0.0,0.0,0.0,0.0,0.0,1.0,0.0,-0.0,-0.0,-0.0,-0.0,-0.0,-0.0,-0.0,-0.609625471048958,
        -1.8210324712466985E-19,-4.8702744413524358E-19,-0.0,-0.84083456430118952,-1.2392259909544564E-20,0.0,0.0,
        0.0,0.0,0.0,0.0,0.0,0.0,1.0,-0.0,-0.0,-0.0,-0.0,-0.0,-0.0,-0.75758587834764846,0.0,-3.3051742928782641E-20,
        5.0906254663616612E-16,0.0,0.0,0.0,0.0,0.0,0.0,0.0,1.0,0.0,-0.0,-0.0,-0.0,-0.0,-0.0,-0.0,-0.0,
        -0.60963041253671413,3.5734093577646393E-19,-0.0,-0.84083847313020632,3.2392852856704325E-20,0.0,0.0,0.0,
        0.0,0.0,0.0,0.0,0.0,1.0,-0.0,-0.0,-0.0,-0.0,-0.0,-0.0,-0.60962843737462846,-6.6103931646927414E-20,-0.0,
        -0.84085610383552944,0.0,0.0,0.0,0.0,0.0,0.0,0.0,0.0,0.0,1.0,-0.0,-0.0,-0.0,-0.0,-0.0,-0.0,-0.0,
        -0.609625471048958,0.0,1.6888683968347326E-16,9.1051623562334923E-20,0.0,0.0,0.0,0.0,0.0,0.0,1.0,-0.0,-0.0,
        -0.0,-0.0,-0.0,-0.0,-0.0,-0.60963041253671413,-4.522365632015879E-20,1.6888856812294667E-16,
        1.2630566289979805E-16,0.0,-1.7867046788823196E-19,0.0,0.0,0.0,0.0,0.0,0.0,1.0,-0.0,-0.0,-0.0,-0.0,-0.0,
        -0.0,-0.0,-0.0,7.481439565165569E-5,-0.45429994164840926,4.8427929846470528E-5,0.84085082053685611,
        -0.00051016981098213191,0.0,0.0,0.0,0.0,0.0,0.0,0.0,0.0,-0.0,-0.0,-0.0,-0.0,-0.0,-0.0,
        0.00018415797916782135,0.00038816816420182129,0.60962237832884059,0.4542999416484092,0.41627806175091842,
        -0.0004141582836222081,-0.60962237832884059,-0.4542999416484092,-0.41627806175091842,0.0,0.0,0.0,0.0,0.0,
        0.0,0.0,0.0,-0.0,-0.0,-0.0,-0.0,-0.0,-0.0,0.00013189937133657251,-0.41628290531231782,0.757562300931841,
        0.55040967557980414,-0.00017606010923842055,0.0,0.0,0.0,0.0,0.0,0.0,0.0,0.0,-0.0,-0.0,-0.0,-0.0,-0.0,-0.0,
        -0.0,0.00022788856259313035,0.00039473384869379729,0.41627862603096338,-0.6096230881794128,
        -0.45430056003742264,-0.41627862603096327,0.0,0.0,0.0,0.0,0.0,0.0,0.0,0.0,1.0,0.0,-0.0,-0.0,-0.0,-0.0,-0.0,
        -0.0,-0.0,8.5975056991699629E-20,0.60962843737462846,1.642350835564962E-19,-3.3777572510500658E-16,
        -2.5261031303621274E-16,0.0,0.0,0.0,0.0,0.0,0.0,0.0,0.0,-0.0,-0.0,-0.0,-0.0,-0.0,-0.0,-0.0,-1.0,
        7.481439565165569E-5,0.45430524726196975,-9.9174781569828316E-5,-0.84085610383552944,0.00051016158613891569,
        0.0,0.0,0.0,0.0,0.0,0.0,0.0,-0.0,-0.0,-0.0,-0.0,-0.0,-0.0,-0.0,0.00013189937133657251,0.41628290531231782,
        -0.00017606010923842055,-0.0001782357389326195,-0.757562300931841,-0.55040967557980436,0.0,0.0,0.0,0.0,0.0,
        0.0,0.0,-0.0,-0.0,-0.0,-0.0,-0.0,-0.0,-0.0,-0.0,-0.45430265350071453,8.5499847267427823E-5,
        -0.55040651377225314,7.846411462241605E-5,0.8408340548111205,-4.8431021786366918E-5,0.0,0.0,0.0,0.0,0.0,0.0,
        0.0,0.0,-0.0,-0.0,-0.0,-0.0,-0.0,-0.0,-0.45430697881955229,8.7898076503418581E-5,-0.55041168721633849,
        0.8408384731302061,-7.8469117928435135E-5,0.0,0.0,0.0,0.0,0.0,0.0,0.0,0.0,-0.0,-0.0,-0.0,-0.0,-0.0,-0.0,
        -0.45430524726196975,0.00010010180270488143,-0.550409675579804,-7.4819295386679732E-5,0.84083690387628529,
        9.9181420037518247E-5,0.0,0.0,0.0,0.0,0.0,0.0,0.0,0.0,-0.0,-0.0,-0.0,-0.0,-0.0,-0.0,-0.0,
        -0.55040651377225314,-8.5505485825257047E-5,0.8408345643011893,4.8427734256521668E-5,0.0001028531289785517,
        0.0,0.0,0.0,0.0,0.0,-0.0,-0.0,-0.0,-0.0,-0.0,0.00015110237018723782,-0.41628054986992113,
        0.00013795452656197144,-8.4707990552849259E-5,0.55040582594762266,0.0,0.0,0.0,0.0,0.0,0.0,0.0,0.0,-0.0,-0.0,
        -0.0,-0.0,-0.0,-0.0,-3.1149970082996928E-20,-1.2630446370897993E-16,-2.3845293855353908E-19,
        0.60962481916553923,-1.8209900679330059E-19,1.6888661273616133E-16,0.0,0.0,0.0,0.0,0.0,0.0,0.0,0.0,-0.0,
        -0.0,-0.0,-0.0,-0.0,-0.0,-1.0,8.54998472674278E-5,7.8464114622416064E-5,0.4543020818309505,
        -4.842792984647046E-5,-0.84085325521465437,0.0005101680221438746,0.0,0.0,0.0,0.0,0.0,-0.0,-0.0,-0.0,-0.0,
        -0.0,0.00015110237018723782,-0.757559413479883,-0.550406513772253,0.00013795452656197138,
        0.41628002822785937,-8.4707990552849354E-5,0.0,0.0,0.0,0.0,0.0,0.0,0.0,-0.0,-0.0,-0.0,-0.0,-0.0,-0.0,-0.0,
        -0.41628450770674136,0.00015561198793193225,0.55041168721633849,-0.0001379545265619716,0.0,0.0,0.0,0.0,0.0,
        0.0,0.0,0.0,-0.0,-0.0,-0.0,-0.0,-0.0,-0.0,-0.41628290531231787,-0.00013189937133657249,0.55040967557980436,
        0.00017606010923842063,0.00017823573893261942,0.0,0.0,0.0,0.0,0.0,0.0,0.0,0.0,-0.0,-0.0,-0.0,-0.0,-0.0,-0.0,
        -0.0,-0.41628054986992108,-0.00015110237018723798,0.55040651377225314,8.4702035317903214E-5,
        0.00018467833523565694,0.0,0.0,0.0,0.0,0.0,-0.0,-0.0,-0.0,-0.0,-0.0,-0.41628450770674136,
        -0.00015561198793193225,0.75756418984348128,0.55041168721633849,0.00010468726281301101,
        0.00013795452656197179,0.0,0.0,0.0,0.0,0.0,0.0,0.0,-0.0,-0.0,-0.0,-0.0,-0.0,-0.0,-0.0,
        -8.803423606264926E-20,0.60963041253671413,3.5734093577646412E-19,3.3777713624589364E-16,
        3.7891698869939418E-16,0.0,0.0,0.0,0.0,0.0,0.0,0.0,0.0,-0.0,-0.0,-0.0,-0.0,-0.0,-0.0,-1.0,
        8.7898076503418486E-5,0.45430697881955218,-7.8464114622416145E-5,-0.84085767302744141,
        0.00051016354941838882,0.0,0.0,0.0,0.0,0.0,-0.0,-0.0,-0.0,-0.0,-0.0,0.00015561198793193222,
        0.41628450770674136,-0.00013795452656197141,-0.75756418984348128,-0.5504116872163386,0.0,0.0,0.0,0.0,0.0,
        0.0,0.0,-0.0,-0.0,-0.0,-0.0,-0.0,-0.0,-0.0,0.60962843737462846,-6.6103931646927414E-20,
        -1.6888786255250324E-16,-1.6423508355649608E-19,-1.2630515651810632E-16,-1.228547004692721E-19,0.0,0.0,0.0,
        0.0,0.0,0.0,0.0,0.0,-0.0,-0.0,-0.0,-0.0,-0.0,-0.0,-1.0,-0.0,0.84087533887700028,1.6889645757588244E-16,
        -6.6103393866630849E-20,0.0,4.5223181965109357E-20,0.0,0.0,0.0,0.0,0.0,0.0,0.0,-0.0,-0.0,-0.0,-0.0,-0.0,
        -0.0,-0.0,-1.0,0.609625471048958,0.0,9.1051623562334923E-20,-1.6888683968347326E-16,-1.2630446370897993E-16,
        0.0,0.0,0.0,0.0,0.0,0.0,-0.0,-0.0,-0.0,-0.0,-0.0,-1.0,0.75758587834764846,0.0,0.84085614120956309,
        -4.9989848646664218E-16,-6.6103349467276677E-20,4.9321661480447027E-20,0.0,6.6103349467276677E-20,0.0,0.0,
        0.0,0.0,0.0,0.0,0.0,0.0,0.0,-0.0,-0.0,-0.0,-0.0,-0.0,-0.0,-0.0,-0.0,-1.0,0.60963041253671413,
        -4.522365632015879E-20,0.0,-1.6888856812294667E-16,-1.7867046788823196E-19,-1.26305662899798E-16,0.0,0.0,
        0.0,0.0,0.0,0.0,0.0,-0.0,-0.0,-0.0,-0.0,-0.0,-0.0,-0.0,-1.0,-7.481439565165569E-5,0.45430524726196975,
        -0.84085610383552944,9.9174781569828492E-5,0.00051016158613891569,0.0001001018027048814,0.0,0.0,0.0,0.0,0.0,
        -0.0,-0.0,-0.0,-0.0,-0.0,-0.0,-0.00018415797916782124,-0.00038816816420182151,0.60962237832884059,
        0.4542999416484092,0.41627806175091842,-0.60962237832884059,-0.4542999416484092,-0.41627806175091842,
        0.00041415828362220767,0.0,0.0,0.0,0.0,0.0,1.0,-0.0,-0.0,-0.0,-0.0,-0.0,-0.0,-0.0,-0.0,
        -0.00013189937133657251,0.41628290531231782,-0.757562300931841,-0.55040967557980436,0.00017606010923842071,
        0.0001782357389326195,0.0,0.0,0.0,0.0,0.0,0.0,0.0,-0.0,-0.0,-0.0,-0.0,-0.0,-0.0,-0.0,-0.0,
        -0.00022788856259313035,-0.00039473384869379729,0.41627862603096338,-0.6096230881794128,
        0.00037493747421003197,0.0,0.0,0.0,0.0,0.0,0.0,0.0,-0.0,-0.0,-0.0,-0.0,-0.0,-0.0,-0.0,0.45430265350071453,
        -8.5499847267427864E-5,-0.84085376462535322,4.8424642574532886E-5,0.00051016694671599048,
        0.00010284562563608354,0.0,0.0,0.0,0.0,-0.0,-0.0,-0.0,-0.0,0.45430697881955229,0.55041168721633871,
        -8.790393854946284E-5,-0.84083847313020632,5.9714664557388114E-5,7.8469117928435325E-5,0.0,0.0,0.0,0.0,0.0,
        0.0,-0.0,-0.0,-0.0,-0.0,-0.0,-0.0,-0.0,-0.0,-0.00015110237018723787,0.41628054986992113,-0.757559413479883,
        8.4702035317903214E-5,-0.55040651377225336,0.00018467833523565724,0.0,0.0,0.0,0.0,0.0,0.0,-0.0,-0.0,-0.0,
        -0.0,-0.0,-0.0,-0.0,0.41628450770674136,-0.00015561198793193225,-0.75756418984348139,0.00010468726281301101,
        -0.55041168721633871,0.00013795452656197179,0.0,0.0,0.0,0.0,0.0,0.0,-0.0,-0.0,-0.0,-0.0,-0.0,-0.0,-0.0,-0.0,
        -1.6888573396344759E-16,-0.84083212995208934,1.753764380417449E-19,-1.1802018608337481E-21,0.0,0.0,0.0,0.0,
        0.0,0.0,0.0,0.0,1.0,0.0,-0.0,-0.0,-0.0,-0.0,-0.0,-0.0,-0.60962237832884059,1.8210324712466982E-19,
        -1.6392577615272447E-19,1.6888575123732502E-16,0.0,0.0,0.0,0.0,0.0,0.0,0.0,-0.0,-0.0,-0.0,-0.0,-0.0,-0.0,
        -0.75756230093184107,3.7331729402847582E-23,-0.84083690387628518,5.53660320073937E-20,
        3.2846577158052279E-19,0.0,0.0,0.0,0.0,0.0,0.0,0.0,1.0,0.0,-0.0,-0.0,-0.0,-0.0,-0.0,-0.0,-0.0,
        -0.60962481916553923,-9.104950339665027E-20,-0.0,4.6369306445630311E-19,-0.84083405481112061,
        -1.1852459228007919E-21,1.0491070505542491E-21,0.0,0.0,0.0,0.0,0.0,0.0,0.0,0.0,1.0,-0.0,-0.0,-0.0,-0.0,-0.0,
        -0.0,-0.75756418984348139,2.1781387555242696E-23,-0.84083847313020632,4.9988181455745605E-16,
        -3.2392852856704325E-20,1.2302723083271699E-19,0.0,0.0,0.0,0.0,0.0,0.0,0.0,0.0,1.0,-0.0,-0.0,-0.0,-0.0,-0.0,
        -0.0,-0.0,-0.60962237832884059,-9.1145916457961507E-20,-3.0930740377156518E-22,1.6888575123732502E-16,
        -4.8686518566049995E-19,0.0,0.0,0.0,0.0,0.0,1.0,-0.0,-0.0,-0.0,-0.0,-0.0,-0.0,-0.0,-0.0,
        -0.60962481916553923,-5.9686710504540159E-20,1.6888661273616133E-16,1.263043082212299E-16,0.0,0.0,0.0,0.0,
        0.0,0.0,0.0,1.0,-0.0,-0.0,-0.0,-0.0,-0.0,-0.0,-0.0,-0.0,7.4819295386679732E-5,-0.55040967557980436,
        0.000510161586138917,0.84083690387628518,-9.9181420037517732E-5,0.0,0.0,0.0,0.0,0.0,0.0,0.0,0.0,-0.0,-0.0,
        -0.0,-0.0,-0.0,-0.0,-0.0,0.00017606010923842057,-0.41627806175091836,8.4707990552849435E-5,
        0.55040260512924977,0.0,0.0,0.0,0.0,0.0,0.0,0.0,0.0,0.0,-0.0,-0.0,-0.0,-0.0,-0.0,-0.0,
        0.00018417146899711557,9.2246400529989555E-7,0.60962172564668826,0.45429936926246767,0.41627753944540197,
        -0.60962172564668826,-0.45429936926246767,-0.41627753944540186,0.0,0.0,0.0,0.0,0.0,0.0,0.0,0.0,1.0,0.0,-0.0,
        -0.0,-0.0,-0.0,-0.0,-0.0,-0.0,-3.3840557120343592E-19,1.2630370373302073E-16,2.7260181487290321E-19,
        0.60962172564668826,-1.6888552398678938E-16,0.0,0.0,0.0,0.0,0.0,0.0,0.0,0.0,0.0,-0.0,-0.0,-0.0,-0.0,-0.0,
        -0.0,-1.0,9.9174781569828235E-5,4.842792984647044E-5,0.45429936926246772,-0.84085082053685589,
        0.00051016981098363212,0.0,0.0,0.0,0.0,0.0,0.0,-0.0,-0.0,-0.0,-0.0,-0.0,8.470203531790335E-5,
        0.00017606010923842057,0.41627806175091836,-0.00018466881149421227,-0.75755643964663877,
        -0.55040329378266917,0.0,0.0,0.0,0.0,0.0,0.0,0.0,-0.0,-0.0,-0.0,-0.0,-0.0,-0.0,8.4707990552849408E-5,
        4.1133666665477103E-7,0.0033259399136323126,-0.75755581033457731,-0.5504026051292501,0.0,0.0,0.0,0.0,0.0,
        0.0,0.0,0.0,-0.0,-0.0,-0.0,-0.0,-0.0,-0.0,-0.0,6.5147957832588729E-20,0.84085610383552933,
        5.0666358765750976E-16,1.0002394461110747E-15,0.0,0.0,0.0,0.0,0.0,0.0,0.0,-0.0,-0.0,-0.0,-0.0,-0.0,-0.0,
        -0.0,-1.0,9.752374880021247E-20,2.69219864857825E-19,0.75755643964663866,-1.2630370373302068E-16,
        -4.8686050246126125E-19,0.0,0.0,0.0,0.0,0.0,0.0,0.0,-0.0,-0.0,-0.0,-0.0,-0.0,-0.0,-1.0,
        7.4819295386679732E-5,0.55040967557980447,-9.9181420037517732E-5,-0.0001001086588859579,
        -0.84083690387628518,0.0,0.0,0.0,0.0,0.0,0.0,0.0,-0.0,-0.0,-0.0,-0.0,-0.0,-0.0,-0.0,-0.0,
        -0.55041168721633849,0.00051016354941819909,-8.790393854946284E-5,0.8408384731302061,5.9714664557388114E-5,
        7.8469117928435325E-5,0.0,0.0,0.0,0.0,0.0,0.0,0.0,-0.0,-0.0,-0.0,-0.0,-0.0,-0.0,-0.0,-0.55040329378266928,
        -4.8427734256521736E-5,-9.9181420037518044E-5,0.84083212995208922,0.00010284859467966867,0.0,0.0,0.0,0.0,
        0.0,-0.0,-0.0,-0.0,-0.0,-0.0,-0.0,-0.45430208183095055,-0.55040582594762288,-7.8469117928435352E-5,
        0.84083405481112039,4.843102178636683E-5,0.0,0.0,0.0,0.0,0.0,0.0,0.0,-0.0,-0.0,-0.0,-0.0,-0.0,-0.0,-0.0,
        -3.1149707480090415E-20,0.75755941347988309,0.0,-1.8210264972536316E-19,-4.8702276280530372E-19,
        -5.090289676538971E-16,0.0,0.0,0.0,0.0,0.0,-0.0,-0.0,-0.0,-0.0,-0.0,-0.0,-1.0,8.5505485825256939E-5,
        7.8469117928435148E-5,0.55040582594762255,-4.843102178636702E-5,-0.84083405481112061,0.0,0.0,0.0,0.0,0.0,
        0.0,0.0,-0.0,-0.0,-0.0,-0.0,-0.0,-0.0,-0.0,-0.4162780617509183,-8.4702035317903322E-5,
        -0.00017606010923842068,0.55040329378266928,0.00018466881149421203,0.0,0.0,0.0,0.0,0.0,-0.0,-0.0,-0.0,-0.0,
        -0.0,-0.0,-0.00010468726281301108,-0.00017823573893261944,0.55040403961997142,-0.0033259399136323117,
        -8.4707990552849354E-5,0.75755581033457708,0.0,0.0,0.0,0.0,0.0,0.0,0.0,-0.0,-0.0,-0.0,-0.0,-0.0,-0.0,-0.0,
        -0.0,-0.41628002822785942,-0.0001379545265619716,0.757558784908481,0.55040582594762277,
        8.4707990552849286E-5,0.0,0.0,0.0,0.0,0.0,0.0,0.0,-0.0,-0.0,-0.0,-0.0,-0.0,-0.0,-0.0,
        -3.9166243175019444E-20,0.75756418984348139,-1.2630566289979805E-16,3.5733825445920967E-19,
        5.0903497598883843E-16,0.0,0.0,0.0,0.0,0.0,0.0,0.0,-0.0,-0.0,-0.0,-0.0,-0.0,-0.0,-1.0,8.7903938549462773E-5,
        0.5504116872163386,-7.8469117928435311E-5,-0.84083847313020632,0.0,0.0,0.0,0.0,0.0,0.0,0.0,-0.0,-0.0,-0.0,
        -0.0,-0.0,-0.0,-0.0,0.75756230093184118,-6.61034858575653E-20,-3.7331729402847559E-23,0.84083690387628518,
        -1.642328857902614E-19,-1.2285307508338753E-19,0.0,0.0,0.0,0.0,0.0,0.0,0.0,-0.0,-0.0,-0.0,-0.0,-0.0,-0.0,
        -0.0,-1.0,-0.0,0.6096230881794128,-8.2110521488695769E-20,-3.1878054029127235E-22,-1.6888599687103994E-16,
        -4.948054548592409E-19,-1.2630387361850009E-16,0.0,0.0,0.0,0.0,0.0,0.0,-0.0,-0.0,-0.0,-0.0,-0.0,-0.0,-1.0,
        -0.0,1.68888545925672E-16,0.84083847313020632,5.090349529564296E-16,-3.2392852856704325E-20,0.0,0.0,0.0,0.0,
        0.0,0.0,0.0,-0.0,-0.0,-0.0,-0.0,-0.0,-0.0,-0.0,-0.0,-1.0,0.75755941347988309,-4.9321788734096E-20,
        -2.8888103944906731E-23,0.0,-5.090289676538971E-16,-4.8702276280530247E-19,0.0,0.0,0.0,0.0,-0.0,-0.0,-0.0,
        -0.0,-0.0,-1.0,0.60962481916553923,-5.9686710504540159E-20,0.0,-1.6888661273616133E-16,
        -1.2630430822122988E-16,0.0,0.0,0.0,0.0,0.0,0.0,0.0,-0.0,-0.0,-0.0,-0.0,-0.0,-0.0,-0.0,-1.0,
        0.75756418984348139,-2.1781387555242688E-23,-4.5223264325215918E-20,0.0,-5.0903497598883764E-16,
        -1.786691272296046E-19,0.0,0.0,0.0,0.0,0.0,-0.0,-0.0,-0.0,-0.0,-0.0,-0.0,-1.0,-7.4819295386679732E-5,
        0.55040967557980447,-0.84083690387628518,9.91814200375179E-5,0.0001001086588859579,0.0,0.0,0.0,0.0,0.0,0.0,
        0.0,-0.0,-0.0,-0.0,-0.0,-0.0,-0.0,-0.0,-0.0,-5.9710851674489663E-5,0.4543005600374227,
        -0.00010010180270488141,-0.84085190118769138,9.7305019763635448E-5,0.0005101684703272578,0.0,0.0,0.0,0.0,
        -0.0,-0.0,-0.0,-0.0,-0.0,-0.0,-0.00018417146899711554,-1.6433908261248681E-6,0.60962172564668826,
        0.45429936926246767,0.41627753944540197,-0.60962172564668826,-0.45429936926246767,-0.41627753944540186,0.0,
        0.0,0.0,0.0,0.0,0.0,0.0,1.0,-0.0,-0.0,-0.0,-0.0,-0.0,-0.0,-0.0,-0.0,-0.0,0.55040651377225325,
        -8.5505485825257E-5,-0.8408345643011893,4.8427734256521695E-5,0.00010285312897855262,0.0,0.0,0.0,0.0,0.0,
        0.0,-0.0,-0.0,-0.0,-0.0,-0.0,-0.0,-0.0,0.45430208183095055,-7.846411462241624E-5,-0.840853255214654,
        4.8427929846470358E-5,0.00051016802214387308,0.0,0.0,0.0,0.0,0.0,0.0,-0.0,-0.0,-0.0,-0.0,-0.0,-0.0,-0.0,
        -0.00013795452656197157,0.41628002822785942,-0.75755878490848116,8.4707990552849259E-5,-0.550405825947623,
        0.0,0.0,0.0,0.0,0.0,0.0,-0.0,-0.0,-0.0,-0.0,-0.0,-0.0,-0.0,-0.0,-0.60962172564668826,1.8211991325743819E-19,
        4.869769891576791E-19,1.6888552398678938E-16,0.0,0.0,0.0,0.0,0.0,0.0,0.0,1.0,0.0,-0.0,-0.0,-0.0,-0.0,-0.0,
        -0.0,-0.0,-0.84083690387628529,1.1099619416141393E-18,-5.5366032007393707E-20,-1.642328857902614E-19,
        -1.2285307508338753E-19,0.0,0.0,0.0,0.0,0.0,0.0,0.0,0.0,1.0,-0.0,-0.0,-0.0,-0.0,-0.0,-0.0,-0.0,
        -0.84083456430118952,4.998780955584154E-16,-3.6929401570902465E-20,9.1051235165092008E-20,
        -4.8702128521147154E-19,0.0,0.0,0.0,0.0,0.0,1.0,-0.0,-0.0,-0.0,-0.0,-0.0,-1.6888571313082695E-16,
        2.0933278467107486E-20,-0.84083212995208934,-8.4419497240682937E-20,9.4703432327985161E-23,
        -4.8685902445272773E-19,0.0,0.0,0.0,0.0,0.0,-0.0,-0.0,-0.0,-0.0,-0.0,-0.0,-0.75755878490848128,
        2.8892611608762185E-23,-5.9686264459664926E-20,-0.84083405481112061,-4.4225931473166894E-22,
        9.10491149162437E-20,0.0,0.0,0.0,0.0,0.0,0.0,0.0,1.0,-0.0,-0.0,-0.0,-0.0,-0.0,-0.0,-0.0,
        -0.60962172564668826,-9.1143806586707121E-20,-2.9022766546388333E-22,1.6888552398678938E-16,
        1.2630354803031406E-16,0.0,0.0,0.0,0.0,0.0,0.0,1.0,-0.0,-0.0,-0.0,-0.0,-0.0,-0.0,-0.0,-0.0,-0.0,
        -0.84085325521465415,-1.6888658327079123E-16,-4.3588336687542244E-20,0.0,9.1049145421375812E-20,0.0,0.0,0.0,
        0.0,0.0,0.0,1.0,-0.0,-0.0,-0.0,-0.0,-0.0,-0.0,-0.550403293782669,9.91814200375178E-5,0.00051016873546545674,
        4.8431021786367026E-5,1.1324499555899527E-6,0.84083161987084709,0.0,0.0,0.0,0.0,0.0,0.0,0.0,0.0,0.0,-0.0,
        -0.0,-0.0,-0.0,-0.0,-0.0,4.8427734256521838E-5,9.91814200375178E-5,0.55040329378266961,
        -0.00010284859467966931,-0.840832129952089,0.0,0.0,0.0,0.0,0.0,0.0,0.0,-0.0,-0.0,-0.0,-0.0,-0.0,-0.0,
        4.932282965723688E-22,0.0,-0.0,2.3390148868998579E-19,0.84083212995208911,-2.0997770285150725E-18,0.0,0.0,
        0.0,0.0,0.0,0.0,0.0,-0.0,-0.0,-0.0,-0.0,-0.0,-0.0,-1.0,4.8431021786366952E-5,2.2909110573910174E-7,
        0.0049960062272682909,-0.840831619870847,0.0,0.0,0.0,0.0,0.0,0.0,0.0,0.0,-0.0,-0.0,-0.0,-0.0,-0.0,-0.0,-0.0,
        9.752354635032987E-20,0.84083690387628507,1.1110082532230706E-18,3.2846577158052289E-19,
        1.2285307508338753E-19,0.0,0.0,0.0,0.0,0.0,0.0,0.0,-0.0,-0.0,-0.0,-0.0,-0.0,-0.0,-0.0,-0.0,-1.0,
        -5.9714664557388216E-5,-0.000100108658885958,0.84083270065149018,-0.0049960062272682874,
        -4.8431021786366918E-5,0.0,0.0,0.0,0.0,0.0,0.0,0.0,-0.0,-0.0,-0.0,-0.0,-0.0,-0.0,-0.0,-0.0,
        6.12256505583179E-19,0.75755878490848116,-1.2630430822122988E-16,-1.8209840926457502E-19,
        -2.0076641711829734E-21,1.184453526596045E-21,0.84083405481112039,0.0,0.0,0.0,0.0,0.0,0.0,0.0,-0.0,-0.0,
        -0.0,-0.0,-0.0,-0.0,-0.0,-1.0,-6.0614409112096141E-20,0.84083456430118952,5.090289676538969E-16,
        -2.7315370549527618E-19,-4.8702128521147357E-19,0.0,0.0,0.0,0.0,0.0,0.0,-0.0,-0.0,-0.0,-0.0,-0.0,-0.0,-0.0,
        -1.0,9.7009564648539721E-21,0.84083847313020621,-7.6367237767394E-16,1.7866871575948447E-19,0.0,0.0,0.0,0.0,
        0.0,0.0,0.0,-0.0,-0.0,-0.0,-0.0,-0.0,-0.0,-0.0,-1.0,0.75755713294087956,-8.2110137308287566E-20,
        -3.7367713213901915E-23,-3.1878155269934057E-22,-5.0902608880363241E-16,-4.9480031627697222E-19,0.0,0.0,0.0,
        0.0,-0.0,-0.0,-0.0,-0.0,-0.0,-0.0,-1.0,-0.0,0.60962172564668826,-9.1143806586707121E-20,
        -2.9022766546388333E-22,-1.6888552398678938E-16,-1.2630354803031404E-16,0.0,0.0,0.0,0.0,0.0,0.0,0.0,-0.0,
        -0.0,-0.0,-0.0,-0.0,-0.0,-0.0,-1.0,-0.0,-3.6929401570902471E-20,-0.0,0.84085325521465415,
        1.6888658327079123E-16,-4.3588336687542244E-20,9.1049145421375812E-20,0.0,0.0,0.0,0.0,0.0,0.0,-0.0,-0.0,
        -0.0,-0.0,-0.0,-0.0,-0.0,-1.0,0.75755878490848128,-5.9686264459664962E-20,-2.8892611608762185E-23,0.0,
        -5.0902816324565257E-16,0.0,0.0,0.0,0.0,0.0,-0.0,-0.0,-0.0,-0.0,-0.0,-0.0,-1.0,0.45429936926246767,
        -4.8431021786366857E-5,0.0049960062272682891,-2.2909110573910145E-7,-0.84083161987084709,0.0,0.0,0.0,0.0,
        0.0,0.0,-0.0,-0.0,-0.0,-0.0,-0.0,-0.0,-0.0,-0.0,-0.0,-8.4707990552849313E-5,-7.5250479866203283E-7,
        0.003325939913632313,-0.75755581033457731,-0.55040260512924977,0.0,0.0,0.0,0.0,0.0,0.0,-0.0,-0.0,-0.0,-0.0,
        -0.0,-0.0,-0.0,-0.0,-0.0,0.55040582594762288,-7.8469117928435392E-5,-0.00051016802214399538,
        -0.0001028531289785522,-0.84083405481112039,4.8431021786366823E-5,0.0,0.0,0.0,0.0,0.0,0.0,-0.0,-0.0,-0.0,
        -0.0,-0.0,-0.0,-0.0,-0.0,-0.840850820536856,1.7234498339055512E-19,-1.1115400945908851E-18,
        1.0327571811693951E-21,0.0,0.0,0.0,0.0,0.0,0.0,0.0,0.0,1.0,0.0,-0.0,-0.0,-0.0,-0.0,-0.0,-0.0,
        -0.84083270065149041,6.4644696919149857E-23,-4.9479871196138011E-19,0.0,0.0,0.0,0.0,0.0,0.0,0.0,1.0,0.0,
        -0.0,-0.0,-0.0,-0.0,-0.0,-0.0,-0.0,-0.84085082053685589,8.7195661360134582E-23,-2.220969953600735E-18,
        -8.4416862202560415E-20,6.0122310366782144E-23,0.0,0.0,0.0,0.0,0.0,0.0,0.0,1.0,-0.0,-0.0,-0.0,-0.0,-0.0,
        -0.0,-0.0,-0.0,-0.75755581033457731,1.6446215595724026E-25,-9.1143508979403014E-20,5.0902442300953653E-16,
        0.0,0.0,0.0,0.0,0.0,0.0,1.0,-0.0,-0.0,-0.0,-0.0,-0.0,-0.0,-0.0,-0.0,0.75755581033457731,
        -9.1143508979403E-20,-1.2721949911164169E-24,-1.6446215595724021E-25,-5.0902442300953574E-16,0.0,0.0,0.0,
        0.0,0.0,-0.0,-0.0,-0.0,-0.0,-0.0,-0.0,-1.0,-0.0,0.840850820536856,1.1115400081964914E-18,
        -8.4416862202560415E-20,3.4597823432971686E-23,0.0,0.0,0.0,0.0,0.0,0.0,-0.0,-0.0,-0.0,-0.0,-0.0,-0.0,-0.0,
        -0.0,-1.0,-0.0,-0.84083161987084709,1.753925793255534E-19,1.1099619109243672E-18,1.0493469223541793E-21,0.0,
        0.0,0.0,0.0,0.0,0.0,0.0,0.0,1.0,0.0,-0.0,-0.0,-0.0,-0.0,-0.0,-0.0,-0.00028983042660450772,
        0.60774185316849594,-0.00032104499842707462,0.45260561554757484,-0.00032423089662980361,0.41470020324647255,
        0.00028983042660450772,-0.60774185316849594,0.00032104499842707462,-0.45260561554757484,
        0.00032423089662980361,-0.41470020324647255,0.0,0.0,0.0,0.0,0.0,0.0,0.0,0.0,0.0,1.0,-0.0,-0.0,-0.0,-0.0,
        -0.0,-0.0,-0.0,-0.0,0.00028983042660450767,0.60771760732198055,-0.00034998845489279349,0.45258306322192471,
        -0.00034322043275703971,0.41467880541713448,-0.60771760732198055,-0.45258306322192471,-0.41467880541713448,
        0.0,0.0,0.0,0.0,0.0,0.0,0.0,0.0,1.0,-0.0,-0.0,-0.0,-0.0,-0.0,-0.0,-0.0,-0.0,-0.60774185316849594,0.0,
        4.9507562444117341E-20,-1.6818696161191519E-16,9.0792333081773271E-20,-1.2581077755555868E-16,0.0,
        -4.9507562444117341E-20,-9.0792333081773247E-20,0.0,0.0,0.0,0.0,0.0,0.0,0.0,0.0,1.0,-0.0,-0.0,-0.0,-0.0,
        -0.0,-0.0,-0.0,-0.0,0.00032104499842707462,-0.60771627901050718,-0.41467763318781908,0.00030990522922148058,
        -0.00020644223064780165,0.60771586837025782,0.45258145885114326,0.414677276341478,-0.45258145885114326,0.0,
        0.0,0.0,0.0,0.0,0.0,0.0,0.0,1.0,-0.0,-0.0,-0.0,-0.0,-0.0,-0.0,-0.0,-0.45260561554757484,
        6.705637981480354E-5,7.4542022764773985E-5,-0.54849096138382369,-6.70627819526479E-5,0.83950908011157221,
        -7.3882932570663252E-5,-7.4549313422904716E-5,0.0,0.0,0.0,0.0,0.0,0.0,0.0,0.0,0.0,-0.0,-0.0,-0.0,-0.0,-0.0,
        -0.0,-0.0,0.00032423089662980361,-0.00024604276486503597,0.607721627098605,-0.00030990522922148096,
        0.45258682574740111,0.41468237096544258,-0.607721627098605,-0.45258682574740111,-0.41468237096544258,0.0,
        0.0,0.0,0.0,0.0,0.0,0.0,0.0,1.0,-0.0,-0.0,-0.0,-0.0,-0.0,-0.0,-0.0,-0.41470020324647261,
        -0.00012282470380310523,0.75586897491059513,-0.00013548671280111892,0.54849096138382369,
        -0.0001366776091554688,0.00012282470380310523,0.00013548671280111892,0.0001366776091554688,0.0,0.0,0.0,0.0,
        0.0,0.0,0.0,0.0,0.0,-0.0,-0.0,-0.0,-0.0,-0.0,-0.0,-0.0,-0.00028983042660450767,0.60771760732198055,
        0.45258306322192471,0.41467880541713448,-0.60771760732198055,0.00034998845489279349,-0.45258306322192471,
        0.00034322043275703966,-0.41467880541713448,0.0,0.0,0.0,0.0,0.0,0.0,0.0,0.0,1.0,-0.0,-0.0,-0.0,-0.0,-0.0,
        -0.0,-0.0,-0.0,0.60774185316849594,0.0,4.9507562444117341E-20,9.0792333081773271E-20,0.0,
        -4.9507562444117341E-20,1.6818696161191519E-16,-9.0792333081773247E-20,1.2581077755555868E-16,0.0,0.0,0.0,
        0.0,0.0,0.0,0.0,0.0,0.0,-0.0,-0.0,-0.0,-0.0,-0.0,-0.0,-0.0,-1.0,-0.00032104499842707462,
        -0.00030990522922148069,0.60771586837025782,0.45258145885114326,0.414677276341478,0.00020644223064780165,
        -0.60771586837025782,-0.414677276341478,0.0,0.0,0.0,0.0,0.0,0.0,0.0,1.0,-0.0,-0.0,-0.0,-0.0,-0.0,-0.0,-0.0,
        -0.0,0.45260561554757484,-6.705637981480354E-5,-7.4542022764774E-5,0.54849096138382369,
        -7.3882932570663252E-5,6.70627819526479E-5,-0.83950908011157221,7.3882932570663252E-5,7.45493134229047E-5,
        0.0,0.0,0.0,0.0,0.0,0.0,0.0,0.0,-0.0,-0.0,-0.0,-0.0,-0.0,-0.0,-0.0,-0.0,-0.00032423089662980361,
        0.607721627098605,0.45258682574740111,0.41468237096544258,0.00024604276486503597,-0.607721627098605,
        0.00030990522922148096,-0.45258682574740111,-0.41468237096544258,0.0,0.0,0.0,0.0,0.0,0.0,0.0,1.0,-0.0,-0.0,
        -0.0,-0.0,-0.0,-0.0,-0.0,-0.0,0.41470020324647261,-0.00012282470380310523,-0.00013548671280111892,
        -0.0001366776091554688,0.00012282470380310523,-0.75586897491059513,0.00013548671280111892,
        -0.54849096138382369,0.0001366776091554688,0.0,0.0,0.0,0.0,0.0,0.0,0.0,0.0,-0.0,-0.0,-0.0,-0.0,-0.0,-0.0,
        -0.0,-0.0,2.9755061164947574E-20,-0.60771760732198044,0.0,1.6817672556185198E-16,1.2334487941221325E-19,
        1.2580321328053461E-16,0.0,0.0,0.0,0.0,0.0,0.0,0.0,1.0,-0.0,-0.0,-0.0,-0.0,-0.0,-0.0,-0.0,-0.0,
        0.00034998845489279343,0.00020644223064780157,0.00036358068816811083,0.60771221968588129,
        0.45257806398899236,0.41467405969907745,-0.60771221968588129,-0.45257806398899236,-0.41467405969907745,0.0,
        0.0,0.0,0.0,0.0,0.0,0.0,0.0,0.0,1.0,-0.0,-0.0,-0.0,-0.0,-0.0,-0.0,-0.0,6.7056379814803486E-5,
        0.83951256820538323,-0.00051559608946867748,-0.0,4.8503929239195573E-5,-0.45257806398899236,
        -0.000515601666520195,0.0,0.0,0.0,0.0,0.0,0.0,0.0,0.0,-0.0,-0.0,-0.0,-0.0,-0.0,-0.0,0.00024604276486503592,
        0.00034322043275703961,0.60771348124036872,-0.00036358068816811078,-0.41467517776491791,0.0,0.0,0.0,0.0,0.0,
        0.0,0.0,1.0,-0.0,-0.0,-0.0,-0.0,-0.0,-0.0,-0.0,0.00012282470380310523,0.54846656219268941,-0.0,
        8.8527830239323147E-5,-0.4146740596990775,0.0,0.0,0.0,0.0,0.0,0.0,0.0,0.0,0.0,-0.0,-0.0,-0.0,-0.0,-0.0,-0.0,
        2.9755061164947574E-20,0.60771760732198044,-0.0,2.0638347693417836E-20,4.8839816704642384E-19,
        2.5160334196432531E-16,0.0,0.0,0.0,0.0,0.0,0.0,0.0,0.0,-0.0,-0.0,-0.0,-0.0,-0.0,-0.0,-1.0,
        6.7056379814803486E-5,0.45258306322192476,-7.9634662796535162E-5,-0.83951256820538323,
        0.00051559608946867759,0.0,0.0,0.0,0.0,0.0,0.0,-0.0,-0.0,-0.0,-0.0,-0.0,-0.0,-0.0,0.00012282470380310523,
        0.41467880541713448,-0.00014643395598641436,-0.00014348094203993502,-0.75584811392108253,
        -0.54846656219268941,0.0,0.0,0.0,0.0,0.0,0.0,0.0,-0.0,-0.0,-0.0,-0.0,-0.0,-0.0,-0.0,-0.0,
        -0.60771627901050718,-4.9506989144368247E-20,-0.83949211543668667,-1.8239303391070821E-19,
        4.8855338534453015E-19,0.0,0.0,0.0,0.0,0.0,0.0,0.0,1.0,-0.0,-0.0,-0.0,-0.0,-0.0,-0.0,-0.83952864747628941,
        3.3637392322383048E-16,0.0,4.9506989144368241E-20,9.0791286551000237E-20,0.0,0.0,-4.9506989144368241E-20,
        -9.0791286551000237E-20,0.0,0.0,0.0,0.0,0.0,0.0,0.0,1.0,-0.0,-0.0,-0.0,-0.0,-0.0,-0.0,-0.607721627098605,
        -1.3618849962265987E-19,-1.2330609381155307E-19,-1.7930100380701504E-19,-1.681784660206933E-16,0.0,0.0,0.0,
        0.0,0.0,0.0,0.0,1.0,-0.0,-0.0,-0.0,-0.0,-0.0,-0.0,-0.0,-0.75586897491059513,1.2581077755555871E-16,
        4.53957044533439E-20,3.3154606304565777E-20,0.0,-4.5395704453343891E-20,0.0,0.0,0.0,0.0,0.0,0.0,0.0,0.0,0.0,
        1.0,-0.0,-0.0,-0.0,-0.0,-0.0,-0.0,-0.0,-0.60771760732198032,3.315489520239038E-20,-1.681767255618521E-16,
        -1.64929553273929E-19,-2.466897588244265E-19,0.0,0.0,0.0,0.0,0.0,0.0,0.0,1.0,-0.0,-0.0,-0.0,-0.0,-0.0,-0.0,
        -0.0,-0.0,-0.60771627901050718,9.9015124888234682E-20,-1.6817618571481423E-16,1.8239417817919302E-19,0.0,
        0.0,0.0,0.0,0.0,0.0,0.0,1.0,-0.0,-0.0,-0.0,-0.0,-0.0,-0.0,-0.0,-0.607721627098605,1.3618849962265987E-19,
        -1.681784660206933E-16,-1.2580449590377112E-16,1.2330609381155307E-19,1.7930100380701509E-19,0.0,0.0,0.0,
        0.0,0.0,0.0,1.0,-0.0,-0.0,-0.0,-0.0,-0.0,-0.0,-0.0,-0.0,7.38757514247254E-5,-0.45258183585658091,
        7.14882463612096E-5,-0.54846526788387562,-4.8508322153241939E-5,0.83949183414948236,0.0,0.0,0.0,0.0,0.0,0.0,
        0.0,0.0,-0.0,-0.0,-0.0,-0.0,-0.0,-0.0,0.00013548671280111887,-0.41467763318781908,0.00013118967602768769,
        -8.85278302393231E-5,0.54846485840188586,0.0,0.0,0.0,0.0,0.0,0.0,0.0,0.0,-0.0,-0.0,-0.0,-0.0,-0.0,-0.0,
        -6.370397382786412E-20,2.5160561935436607E-16,1.7976260569382681E-19,0.60771586837025771,0.0,
        1.6817602023351553E-16,0.0,0.0,0.0,0.0,0.0,0.0,0.0,0.0,-0.0,-0.0,-0.0,-0.0,-0.0,-0.0,-1.0,
        7.1488246361209635E-5,0.45258145885114326,-4.8503929239195519E-5,-0.839511404940604,0.00051560018494341568,
        0.0,0.0,0.0,0.0,0.0,-0.0,-0.0,-0.0,-0.0,-0.0,-0.452586825747401,7.4542022764773945E-5,-0.54847065730144762,
        0.83949563162130481,-7.1495079606071117E-5,0.0,0.0,0.0,0.0,0.0,0.0,0.0,0.0,-0.0,-0.0,-0.0,-0.0,-0.0,-0.0,
        -0.45258306322192471,7.8123623135183722E-5,-0.54846656219268941,-6.7062781952647926E-5,0.83949299775843811,
        7.9642715680471464E-5,0.0,0.0,0.0,0.0,0.0,0.0,0.0,0.0,-0.0,-0.0,-0.0,-0.0,-0.0,-0.0,-0.0,
        -0.45258183585658085,-0.54846526788387551,-7.3882932570663293E-5,0.83949211543668689,4.8506315421467726E-5,
        7.3636376402749123E-5,0.0,0.0,0.0,0.0,0.0,-0.0,-0.0,-0.0,-0.0,-0.0,-0.452586825747401,5.7353204127738534E-5,
        7.1488246361209526E-5,-0.54847065730144762,-7.4549313422904716E-5,0.83949563162130481,0.0,0.0,0.0,0.0,0.0,
        0.0,0.0,-0.0,-0.0,-0.0,-0.0,-0.0,-0.0,-0.0,0.0001366776091554688,-0.41468237096544247,
        -0.00013118967602768778,0.54847065730144773,0.0,0.0,0.0,0.0,0.0,0.0,0.0,0.0,-0.0,-0.0,-0.0,-0.0,-0.0,-0.0,
        -7.9990129001169258E-20,0.607721627098605,0.0,1.6817846602069321E-16,1.2580449590377107E-16,0.0,0.0,0.0,0.0,
        0.0,0.0,0.0,0.0,-0.0,-0.0,-0.0,-0.0,-0.0,-0.0,-1.0,7.4542022764773972E-5,0.45258682574740106,
        -7.1488246361209486E-5,-0.83951520168604254,0.000515596671407826,0.0,0.0,0.0,0.0,0.0,-0.0,-0.0,-0.0,-0.0,
        -0.0,0.0001366776091554688,0.41468237096544247,-0.00010492369622770082,-0.00013118967602768778,
        -0.75585156501645778,-0.54847065730144773,0.0,0.0,0.0,0.0,0.0,0.0,0.0,-0.0,-0.0,-0.0,-0.0,-0.0,-0.0,-0.0,
        -0.41467880541713448,-0.00012282470380310526,0.54846656219268952,0.00014643395598641431,
        0.0001434809420399348,0.0,0.0,0.0,0.0,0.0,0.0,0.0,0.0,-0.0,-0.0,-0.0,-0.0,-0.0,-0.0,-0.0,-0.414677633187819,
        -0.00013548671280111889,0.54846526788387573,8.8524154773604152E-5,0.00013469943293139259,0.0,0.0,0.0,0.0,
        0.0,-0.0,-0.0,-0.0,-0.0,-0.0,-0.41468237096544253,-0.00013667760915546878,0.54847065730144762,
        0.0001049236962277008,0.00013118967602768775,0.0,0.0,0.0,0.0,0.0,0.0,0.0,-0.0,-0.0,-0.0,-0.0,-0.0,-0.0,-0.0,
        -2.9755061164947574E-20,0.60771760732198044,0.0,-1.6817672556185198E-16,-1.233448794122132E-19,
        -1.2580321328053463E-16,0.0,0.0,0.0,0.0,0.0,0.0,0.0,0.0,-0.0,-0.0,-0.0,-0.0,-0.0,-0.0,-0.0,-1.0,
        -0.00020643328051976208,-0.00034998845489279343,0.60771263100274964,0.00032311337431655543,
        -0.41467441716242903,0.0,0.0,0.0,0.0,0.0,0.0,1.0,-0.0,-0.0,-0.0,-0.0,-0.0,-0.0,-0.0,-0.0,
        -6.7056379814803486E-5,0.45258306322192476,-0.83951256820538323,7.9634662796535162E-5,7.8123623135183722E-5,
        0.00051559608946867759,0.0,0.0,0.0,0.0,0.0,-0.0,-0.0,-0.0,-0.0,-0.0,-0.0,-0.00024604276486503592,
        -0.00034322043275703955,-0.0002064422306478016,-0.00032311337431655576,0.60771221968588129,
        0.45257806398899236,0.41467405969907745,-0.60771221968588129,-0.41467405969907745,0.0,0.0,0.0,0.0,0.0,0.0,
        0.0,1.0,-0.0,-0.0,-0.0,-0.0,-0.0,-0.0,-0.0,-0.0,-0.0,-0.00012282470380310523,0.41467880541713448,
        -0.75584811392108253,0.00014643395598641436,-0.54846656219268941,0.00014348094203993497,0.0,0.0,0.0,0.0,0.0,
        0.0,0.0,-0.0,-0.0,-0.0,-0.0,-0.0,-0.0,-0.0,-0.0,0.60771627901050718,9.9015124888234682E-20,
        1.8239417817919302E-19,1.6817618571481423E-16,0.0,1.2580280967718299E-16,0.0,0.0,0.0,0.0,0.0,-0.0,-0.0,-0.0,
        -0.0,-0.0,-1.0,0.83952864747628941,-3.3637392322383053E-16,0.0,4.9506989144368241E-20,
        9.0791286551000237E-20,0.0,-4.9506989144368241E-20,-9.0791286551000237E-20,0.0,0.0,0.0,0.0,0.0,0.0,0.0,-0.0,
        -0.0,-0.0,-0.0,-0.0,-0.0,-0.0,-1.0,0.607721627098605,1.3618849962265987E-19,1.2330609381155307E-19,
        1.7930100380701509E-19,1.681784660206933E-16,1.2580449590377112E-16,0.0,0.0,0.0,0.0,0.0,0.0,0.0,-0.0,-0.0,
        -0.0,-0.0,-0.0,-0.0,-0.0,-1.0,0.75586897491059513,-1.2581077755555871E-16,4.53957044533439E-20,
        3.3154606304565777E-20,0.0,0.0,0.0,0.0,0.0,0.0,0.0,0.0,-0.0,-0.0,-0.0,-0.0,-0.0,-0.0,-1.0,
        -7.38757514247254E-5,0.45258183585658091,4.850192273613149E-5,-0.83951168616294036,7.3628717755583559E-5,
        0.00051559955622434669,0.0,0.0,0.0,0.0,-0.0,-0.0,-0.0,-0.0,-0.00013548671280111887,-0.00013118967602768775,
        0.414677276341478,8.852783023932312E-5,-0.75584662495331045,-0.54846485840188586,0.0,0.0,0.0,0.0,0.0,0.0,
        -0.0,-0.0,-0.0,-0.0,-0.0,-0.0,-0.0,-0.0,0.452586825747401,-7.4542022764773945E-5,5.7353204127738534E-5,
        -0.83951520168604254,7.1488246361209567E-5,0.00051559667140782691,0.0,0.0,0.0,0.0,0.0,0.0,-0.0,-0.0,-0.0,
        -0.0,-0.0,-0.0,-0.0,-0.0001366776091554688,0.41468237096544247,0.00010492369622770083,-0.75585156501645778,
        0.00013118967602768764,-0.54847065730144773,0.0,0.0,0.0,0.0,0.0,0.0,-0.0,-0.0,-0.0,-0.0,-0.0,-0.0,-0.0,-0.0,
        -8.246374572135012E-20,9.8108818261083368E-20,-0.83950898205466618,-8.9882277746204806E-26,
        4.985436410395924E-16,0.0,0.0,0.0,0.0,0.0,0.0,0.0,0.0,1.0,-0.0,-0.0,-0.0,-0.0,-0.0,-0.0,
        2.9754765431896156E-20,-0.83951256820538334,0.0,0.0,4.9854995011635195E-16,0.0,0.0,0.0,0.0,0.0,0.0,-0.0,
        -0.0,-0.0,-0.0,-0.0,-0.0,8.8392842585362538E-20,-1.8501731911831992E-19,9.8109375285541218E-20,
        -0.60771221968588129,1.6817447504922767E-16,0.0,0.0,0.0,0.0,0.0,0.0,0.0,0.0,1.0,-0.0,-0.0,-0.0,-0.0,-0.0,
        -0.0,-0.0,6.7062781952647967E-5,0.839492997758438,-0.0,0.00051560103798285685,4.8508322153242075E-5,
        -0.0049959693296679321,1.1481092117693212E-6,0.0,0.0,0.0,0.0,0.0,0.0,0.0,0.0,0.0,-0.0,-0.0,-0.0,-0.0,-0.0,
        -0.0,0.00010492369622770083,0.0001434809420399351,8.8527830239323147E-5,0.00013470903175427876,
        0.4146740596990775,-0.75584347736259117,-0.54846116837011871,0.0,0.0,0.0,0.0,0.0,0.0,0.0,0.0,-0.0,-0.0,-0.0,
        -0.0,-0.0,-0.0,-0.0,2.9754765431896156E-20,0.83951256820538334,0.0,0.0,-4.9854995011635195E-16,0.0,0.0,0.0,
        0.0,0.0,0.0,-0.0,-0.0,-0.0,-0.0,-0.0,-0.0,-0.0,-1.0,6.7062781952647967E-5,0.54846656219268952,
        -7.9642715680471464E-5,-7.8131577710013753E-5,-0.839492997758438,0.0,0.0,0.0,0.0,0.0,0.0,0.0,-0.0,-0.0,-0.0,
        -0.0,-0.0,-0.0,-0.0,-0.0,-0.60771586837025771,5.9508718159756055E-20,-4.8884752457005644E-19,
        -9.1195009050586689E-20,-1.6817602023351548E-16,0.0,0.0,0.0,0.0,0.0,0.0,0.0,1.0,-0.0,-0.0,-0.0,-0.0,-0.0,
        -0.0,-0.0,-4.625701589801718E-23,-9.0791286551000225E-20,-0.83949563162130469,0.0,0.0,0.0,0.0,0.0,0.0,0.0,
        0.0,0.0,1.0,-0.0,-0.0,-0.0,-0.0,-0.0,-0.0,-0.8395090801115721,1.1104954790887438E-18,
        -3.3154532651703232E-20,4.950692740610004E-20,9.0791173929120774E-20,3.3154532651703232E-20,
        -4.950692740610004E-20,-9.0791173929120762E-20,0.0,0.0,0.0,0.0,0.0,0.0,0.0,0.0,0.0,1.0,-0.0,-0.0,-0.0,-0.0,
        -0.0,-0.0,-0.0,0.0,-2.4668692135355611E-19,-0.83949299775843789,-6.2635751390691967E-21,
        -1.64927269518349E-19,0.0,0.0,0.0,0.0,0.0,0.0,0.0,0.0,1.0,-0.0,-0.0,-0.0,-0.0,-0.0,-0.0,-0.0,
        -3.1490119814551088E-23,-0.83949211543668667,4.2469420815797451E-20,1.8239303391070821E-19,
        -4.8855338534452948E-19,0.0,0.0,0.0,0.0,0.0,1.0,-0.0,-0.0,-0.0,-0.0,-0.0,-0.83951520168604232,
        -4.625701589801718E-23,9.0791286551000225E-20,-4.9855482999028193E-16,6.1652571145841663E-20,0.0,0.0,0.0,
        0.0,0.0,0.0,0.0,1.0,-0.0,-0.0,-0.0,-0.0,-0.0,-0.0,-0.83949563162130458,1.1104953763821025E-18,
        6.683190108752474E-22,1.2330504017361608E-19,0.0,0.0,0.0,0.0,0.0,0.0,0.0,0.0,1.0,-0.0,-0.0,-0.0,-0.0,-0.0,
        -0.0,-0.0,-0.60771263100274964,-9.1103604592422571E-20,1.6492955327392894E-19,-4.8839816704642317E-19,0.0,
        0.0,0.0,0.0,0.0,0.0,1.0,-0.0,-0.0,-0.0,-0.0,-0.0,-0.0,-0.0,-0.0,-0.60771348124036884,-0.83950981017513349,
        -8.20210993821808E-20,2.46686921353556E-19,-4.9854515452033152E-16,0.0,0.0,0.0,0.0,0.0,0.0,1.0,-0.0,-0.0,
        -0.0,-0.0,-0.0,-0.0,-0.0,-0.60771586837025771,-5.9508718159756067E-20,-1.6817602023351548E-16,
        -1.2580268781145876E-16,9.1195009050586689E-20,0.0,0.0,0.0,0.0,0.0,0.0,1.0,-0.0,-0.0,-0.0,-0.0,-0.0,-0.0,
        -0.0,-0.0,0.00013118967602768769,0.00013469943293139243,0.414677276341478,-8.85278302393231E-5,
        -0.75584662495331045,-0.54846485840188586,0.0,0.0,0.0,0.0,0.0,0.0,0.0,-0.0,-0.0,-0.0,-0.0,-0.0,-0.0,-0.0,
        1.8151062270724029E-19,0.83951140494060406,-1.6817602023351545E-16,0.0,0.0,0.0,0.0,0.0,0.0,0.0,-0.0,-0.0,
        -0.0,-0.0,-0.0,-1.0,7.3882932570663347E-5,7.1495079606071347E-5,0.54846485840188541,-4.8508322153242115E-5,
        -0.83949183414948259,0.0,0.0,0.0,0.0,0.0,0.0,0.0,-0.0,-0.0,-0.0,-0.0,-0.0,-0.0,-0.0,-0.45257924052569581,
        -5.73532041277385E-5,-7.8123623135183614E-5,0.83950981017513371,-0.00051560065177808285,
        8.2669047804172151E-5,0.0,0.0,0.0,0.0,0.0,-0.0,-0.0,-0.0,-0.0,-0.0,-0.0,-0.0,-0.45258145885114337,
        -0.54846485840188586,-7.1495079606071212E-5,0.83949183414948259,4.8508322153242129E-5,0.0,0.0,0.0,0.0,0.0,
        0.0,0.0,-0.0,-0.0,-0.0,-0.0,-0.0,-0.0,-0.0,-8.7176738319430579E-20,0.83951520168604243,
        -1.6817846602069328E-16,0.0,0.0,0.0,0.0,0.0,0.0,0.0,-0.0,-0.0,-0.0,-0.0,-0.0,-1.0,0.75585156501645778,
        -1.2580449590377104E-16,-1.7929917369533893E-19,-6.96516636356949E-22,0.83949563162130481,
        -6.1652520086808E-20,0.0,0.0,0.0,0.0,0.0,0.0,0.0,-0.0,-0.0,-0.0,-0.0,-0.0,-0.0,-0.0,-1.0,
        7.454931342290477E-5,0.54847065730144728,-5.7358524655122212E-5,-7.1495079606071239E-5,-0.83949563162130492,
        0.0,0.0,0.0,0.0,0.0,0.0,0.0,-0.0,-0.0,-0.0,-0.0,-0.0,-0.0,-0.0,-0.41467517776491786,-0.00010492369622770092,
        -0.00014348094203993486,0.54846243479694534,0.00015236510263377253,0.0,0.0,0.0,0.0,0.0,0.0,0.0,-0.0,-0.0,
        -0.0,-0.0,-0.0,-0.0,-0.0,-0.41467727634147794,-0.0001311896760276878,0.548464858401886,8.85278302393231E-5,
        0.0,0.0,0.0,0.0,0.0,0.0,0.0,-0.0,-0.0,-0.0,-0.0,-0.0,-0.0,-0.0,-8.839284258536255E-20,0.60771348124036884,
        1.8501731911831983E-19,-9.8109375285541218E-20,-1.6817447504922767E-16,-1.2580154888538883E-16,0.0,0.0,0.0,
        0.0,0.0,0.0,0.0,-0.0,-0.0,-0.0,-0.0,-0.0,-0.0,-0.0,-0.0,-1.0,-2.975480007865129E-20,0.75584811392108275,0.0,
        0.0,-5.0668078577586268E-16,-1.2334362658056649E-19,0.0,0.0,0.0,0.0,0.0,0.0,-0.0,-0.0,-0.0,-0.0,-0.0,-0.0,
        -0.0,-1.0,-0.00014643395598641445,-8.8527830239323147E-5,-0.00015236510263377253,0.4146740596990775,
        -0.54846116837011871,0.0,0.0,0.0,0.0,0.0,0.0,-0.0,-0.0,-0.0,-0.0,-0.0,-0.0,-0.0,-0.0,-0.0,
        -5.7353204127738527E-5,0.45257924052569587,-7.8123623135183655E-5,-0.8395098101751336,8.2669047804172151E-5,
        0.00051560065177708408,0.0,0.0,0.0,0.0,-0.0,-0.0,-0.0,-0.0,-0.0,-0.0,-6.7062781952647967E-5,
        0.54846656219268952,-0.839492997758438,7.9642715680471464E-5,7.81315777100136E-5,0.0,0.0,0.0,0.0,0.0,0.0,
        0.0,-0.0,-0.0,-0.0,-0.0,-0.0,-0.0,-0.0,-0.0,-0.00010492369622770084,-0.00014348094203993505,
        0.41467517776491797,-0.75584455578182586,0.0001523651026337728,-0.54846243479694468,0.0,0.0,0.0,0.0,0.0,
        -0.0,-0.0,-0.0,-0.0,-0.0,-0.0,-0.0,0.60771586837025771,-5.9508718159756067E-20,9.1195009050586689E-20,
        1.6817602023351548E-16,1.2580268781145876E-16,0.0,0.0,0.0,0.0,0.0,0.0,0.0,-0.0,-0.0,-0.0,-0.0,-0.0,-0.0,
        -0.0,-1.0,0.75584698353565438,3.6297211588305579E-20,-1.258027775726083E-16,1.8239326798807447E-19,0.0,0.0,
        0.0,0.0,0.0,0.0,-0.0,-0.0,-0.0,-0.0,-0.0,-1.0,0.8395090801115721,1.1099594411114691E-18,
        -3.3154532651703232E-20,4.950692740610004E-20,9.0791173929120774E-20,3.3154532651703232E-20,
        -4.950692740610004E-20,-9.0791173929120762E-20,0.0,0.0,0.0,0.0,0.0,0.0,0.0,0.0,-0.0,-0.0,-0.0,-0.0,-0.0,
        -0.0,-0.0,-0.0,-1.0,-7.1488246361209608E-5,0.4525814588511432,4.8503929239195519E-5,-0.83951140494060417,
        0.00051560018494391658,0.0,0.0,0.0,0.0,0.0,0.0,-0.0,-0.0,-0.0,-0.0,-0.0,-0.0,-0.0,-7.3882932570663347E-5,
        0.54846526788387562,4.8506315421467529E-5,-0.83949211543668678,7.36363764027489E-5,0.0,0.0,0.0,0.0,0.0,0.0,
        -0.0,-0.0,-0.0,-0.0,-0.0,-0.0,-0.0,0.54847065730144762,-7.454931342290473E-5,5.7358524655122233E-5,
        -0.83949563162130481,7.1495079606071144E-5,0.0,0.0,0.0,0.0,0.0,0.0,-0.0,-0.0,-0.0,-0.0,-0.0,-0.0,-0.0,-0.0,
        2.9754733575446928E-20,-0.839492997758438,-4.9854995011635155E-16,0.0,0.0,0.0,0.0,0.0,0.0,0.0,0.0,0.0,1.0,
        -0.0,-0.0,-0.0,-0.0,-0.0,-0.0,-0.0,5.6433356177770327E-20,-7.00966397529624E-22,0.60771221968588141,
        1.6817447504922767E-16,1.2580154888538883E-16,0.0,0.0,0.0,0.0,0.0,0.0,0.0,0.0,0.0,-0.0,-0.0,-0.0,-0.0,-0.0,
        -0.0,-1.0,4.8503929239195573E-5,7.3634033153687213E-5,0.45257806398899231,-0.83950898205466606,
        0.000515601666520195,0.0,0.0,0.0,0.0,0.0,0.0,-0.0,-0.0,-0.0,-0.0,-0.0,-1.6262870258933998E-19,
        -1.6817464083486873E-16,4.9240506899104478E-20,0.8395089820546664,-1.1115503907899016E-18,0.0,0.0,0.0,0.0,
        0.0,0.0,-0.0,-0.0,-0.0,-0.0,-0.0,-1.0,5.7358524655122206E-5,7.8131577710013631E-5,0.54846243479694479,
        4.8508322153242088E-5,0.004995969329667933,-0.83948941084011008,0.0,0.0,0.0,0.0,0.0,0.0,0.0,0.0,-0.0,-0.0,
        -0.0,-0.0,-0.0,-0.0,-0.0,2.9754733575446928E-20,0.839492997758438,-2.5322003579499064E-16,0.0,
        1.2334330862335358E-19,0.0,0.0,0.0,0.0,0.0,0.0,0.0,-0.0,-0.0,-0.0,-0.0,-0.0,-0.0,-0.0,-0.0,-1.0,
        4.850631542146761E-5,7.9642715680471531E-5,0.54846157851902466,-7.3641691938526E-5,-0.839489692551959,0.0,
        0.0,0.0,0.0,0.0,0.0,0.0,-0.0,-0.0,-0.0,-0.0,-0.0,-0.0,5.9508025155671187E-20,-3.7944716262115873E-23,
        -4.88843264703953E-19,-0.83949183414948236,-1.0685174091063236E-21,-1.8238887367955244E-19,0.0,0.0,0.0,0.0,
        0.0,0.0,0.0,0.0,1.0,-0.0,-0.0,-0.0,-0.0,-0.0,-0.0,-0.83951140494060383,-3.7944716262115873E-23,
        -5.9508025155671235E-20,-4.9854794748204026E-16,9.119449206614489E-20,0.0,0.0,0.0,0.0,0.0,0.0,1.0,-0.0,-0.0,
        -0.0,-0.0,-0.0,-0.0,1.1104954242848737E-18,0.0,-0.0,-0.83950898205466606,-9.1080341125208536E-20,
        1.0218805379139446E-24,0.0,0.0,0.0,0.0,0.0,0.0,1.0,-0.0,-0.0,-0.0,-0.0,-0.0,-0.0,-0.0,-0.83949183414948236,
        1.110495398303592E-18,-6.0094685994419228E-22,1.8238887367955241E-19,0.0,0.0,0.0,0.0,0.0,0.0,0.0,1.0,-0.0,
        -0.0,-0.0,-0.0,-0.0,-0.0,-0.0,-0.60771221968588141,-9.1080860224906571E-20,1.0218648896758904E-24,
        -1.6817447504922772E-16,-1.2580154888538883E-16,0.0,0.0,0.0,0.0,0.0,0.0,1.0,-0.0,-0.0,-0.0,-0.0,-0.0,-0.0,
        -0.0,-0.0,-0.0,0.75584662495331045,-3.7740806343437641E-16,-9.1194553892523224E-20,1.6475704522131309E-21,
        0.83949183414948247,0.0,0.0,0.0,0.0,0.0,0.0,0.0,-0.0,-0.0,-0.0,-0.0,-0.0,-0.0,-0.0,-1.0,
        0.00051560065177795838,-5.7358524655122192E-5,-7.81315777100136E-5,0.83949023913090359,
        -0.0049959693296679373,1.1481092117723822E-6,-4.8508322153242E-5,0.0,0.0,0.0,0.0,0.0,0.0,0.0,-0.0,-0.0,-0.0,
        -0.0,-0.0,-0.0,-0.0,-0.0,-0.45257806398899231,-4.8503929239195492E-5,-8.2669047804172476E-5,
        0.83950898205466629,-0.00051560166652169328,0.0,0.0,0.0,0.0,0.0,0.0,-0.0,-0.0,-0.0,-0.0,-0.0,-0.0,-0.0,-0.0,
        -0.41467405969907745,-8.852783023932331E-5,-0.00015236510263377218,0.54846116837011893,0.0,0.0,0.0,0.0,0.0,
        0.0,0.0,-0.0,-0.0,-0.0,-0.0,-0.0,-0.0,-0.0,-0.0,-3.6975241712266472E-20,0.755844555781826,
        1.3769388015871068E-19,1.2580195959048207E-16,0.0,0.0,0.0,0.0,0.0,0.0,-0.0,-0.0,-0.0,-0.0,-0.0,-0.0,-0.0,
        -1.0,-2.9754733575446928E-20,0.839492997758438,-2.5322003579499064E-16,0.0,-1.2334330862335355E-19,0.0,0.0,
        0.0,0.0,0.0,0.0,0.0,-0.0,-0.0,-0.0,-0.0,-0.0,-0.0,-0.0,-0.0,-1.0,0.45257806398899236,-0.0,
        -4.850631542146761E-5,-7.9642715680471531E-5,0.54846157851902466,-0.839489692551959,0.0,0.0,0.0,0.0,0.0,0.0,
        -0.0,-0.0,-0.0,-0.0,-0.0,-0.0,-0.0,-0.0,-5.7358524655122206E-5,0.548462434796945,-7.8131577710013631E-5,
        -0.83949023913090348,8.2677296121898793E-5,0.0,0.0,0.0,0.0,0.0,-0.0,-0.0,-0.0,-0.0,-0.0,-0.0,-0.0,
        4.2469420815797463E-20,0.83949183414948236,-6.0094685994419191E-22,-1.110495398303592E-18,
        1.8238887367955244E-19,0.0,0.0,0.0,0.0,0.0,0.0,-0.0,-0.0,-0.0,-0.0,-0.0,-0.0,-0.0,-0.0,-1.0,
        0.83949563162130469,1.1099596201273517E-18,6.683190108752475E-22,1.2330504017361606E-19,0.0,0.0,0.0,0.0,0.0,
        0.0,0.0,-0.0,-0.0,-0.0,-0.0,-0.0,-0.0,-0.0,-0.0,-1.0,-7.149507960607132E-5,0.54846485840188608,
        -7.3636376402749177E-5,-0.00051560018494413527,4.8508322153241933E-5,-0.83949183414948236,0.0,0.0,0.0,0.0,
        0.0,0.0,-0.0,-0.0,-0.0,-0.0,-0.0,-0.0,-0.0,-0.0,9.811099909019153E-20,-0.83948969255195927,
        -5.9470437978074124E-22,-1.1104954909955548E-18,4.8839345513964346E-19,0.0,0.0,0.0,0.0,0.0,0.0,0.0,0.0,1.0,
        -0.0,-0.0,-0.0,-0.0,-0.0,-0.0,8.5051560381848912E-20,-5.5577944565858811E-19,0.0,0.0,0.0,0.0,0.0,0.0,0.0,
        0.0,0.0,1.0,-0.0,-0.0,-0.0,-0.0,-0.0,-0.0,-1.0,7.7873197452969825E-20,2.803986063763796E-19,
        6.4296063569359765E-22,0.83948941084011031,3.330933417383221E-18,0.0,0.0,0.0,0.0,0.0,0.0,0.0,0.0,-0.0,-0.0,
        -0.0,-0.0,-0.0,-0.0,-0.0,-1.0,3.3215168474146733E-20,-1.0697498708079556E-21,0.83949023913090381,0.0,0.0,
        0.0,0.0,0.0,0.0,0.0,0.0,-0.0,-0.0,-0.0,-0.0,-0.0,-0.0,-0.0,-1.0,-8.8392085258418591E-20,0.83949023913090348,
        -1.109959330793548E-18,5.7702323571187137E-22,0.0,0.0,0.0,0.0,0.0,0.0,-0.0,-0.0,-0.0,-0.0,-0.0,-0.0,-0.0,
        -1.0,-9.811099909019153E-20,5.9470437978074124E-22,0.83948941084011031,1.1104955074523147E-18,0.0,0.0,0.0,
        0.0,0.0,0.0,-0.0,-0.0,-0.0,-0.0,-0.0,-0.0,-0.0,-0.0,-0.0,-1.0,4.1039746089312351E-20,-0.83948941084011031,
        -1.1010645961606569E-21,-1.1104955074523147E-18,0.0,0.0,0.0,0.0,0.0,0.0,0.0,0.0,0.0,1.0,-0.0,-0.0,-0.0,-0.0,
        -0.0,-0.0];
    Explicit_b_G: ARRAY [0..249] OF LREAL := [0.0,0.0,140.328,-0.066712260924210731,-0.06481259658265906,136.328,
        70.09208224196523,-0.049529802998884785,-0.04991060377936854,68.093414975642048,46.672260105606064,
        -0.036349978139805554,-0.037442373571299752,45.340877278654531,-10.0,0.0047540234966799736,
        0.0066558326400829385,-14.0,-4.9948750243689952,0.0035295737841973653,0.005125494783985384,
        -6.9927513765256482,-3.3259406608521505,0.0025903581708429926,0.0038450885364576352,-4.6562135577516246,
        140.32799999999997,136.32800000000003,140.328,-0.0667725858975615,140.328,68.077973963187517,
        140.32799999999997,-0.066766750479010858,140.328,45.312597285515771,140.328,-13.999999999999998,
        140.32799999999997,-7.0081863352279727,140.32799999999997,-4.684485232538492,70.07529315333116,136.328,
